   VAR
      sa_Parameter { ExternalAccessible := 'False'; ExternalVisible := 'False'; ExternalWritable := 'False'; S7_SetPoint := 'False'} : Array[1..16] of "UDT_VfdSinaParameterUser";   // Structure with parameters
      sa_ParameterEmpty { ExternalAccessible := 'False'; ExternalVisible := 'False'; ExternalWritable := 'False'; S7_SetPoint := 'False'} : Array[1..16] of "UDT_VfdSinaParameterUser";   // Empty structure
      sa_ParameterToCompare { ExternalAccessible := 'False'; ExternalVisible := 'False'; ExternalWritable := 'False'; S7_SetPoint := 'False'} : Array[1..16] of "UDT_VfdSinaParameterUser";   // Structure with parameters to compare
      sFB_SinaParaInstance {InstructionName := 'SinaPara'; LibVersion := '1.1'; ExternalAccessible := 'False'; ExternalVisible := 'False'; ExternalWritable := 'False'; S7_SetPoint := 'False'} : SinaPara;   // Write/read parameters to/from VFD
      sR_TRIG_StartJob {InstructionName := 'R_TRIG'; LibVersion := '1.0'; ExternalAccessible := 'False'; ExternalVisible := 'False'; ExternalWritable := 'False'; S7_SetPoint := 'False'} : R_TRIG;   // Bit for start trigger for rising edge
      sR_TRIG_Time {InstructionName := 'R_TRIG'; LibVersion := '1.0'; ExternalAccessible := 'False'; ExternalVisible := 'False'; ExternalWritable := 'False'; S7_SetPoint := 'False'} : R_TRIG;   // Bit for trigger for time couting
      sR_TRIG_DelayTime {InstructionName := 'R_TRIG'; LibVersion := '1.0'; ExternalAccessible := 'False'; ExternalVisible := 'False'; ExternalWritable := 'False'; S7_SetPoint := 'False'} : R_TRIG;   // Bit for trigger for time couting
      sF_TRIG_CancelJob {InstructionName := 'F_TRIG'; LibVersion := '1.0'; ExternalAccessible := 'False'; ExternalVisible := 'False'; ExternalWritable := 'False'; S7_SetPoint := 'False'} : F_TRIG;   // Bit for start trigger for falling edge
      sa_Status { ExternalAccessible := 'False'; ExternalVisible := 'False'; ExternalWritable := 'False'} : Struct   // Parametrization status
         StepNr { ExternalAccessible := 'False'; ExternalVisible := 'False'; ExternalWritable := 'False'} : Int;   // The number of the current step
         StepNrError { ExternalAccessible := 'False'; ExternalVisible := 'False'; ExternalWritable := 'False'} : Int;   // The number of the step in witch the error occurred
         ParameterNrError { ExternalAccessible := 'False'; ExternalVisible := 'False'; ExternalWritable := 'False'} : Int;   // The number of the parameter in witch the error occurred
         ResponseValueError { ExternalAccessible := 'False'; ExternalVisible := 'False'; ExternalWritable := 'False'} : Bool;   // Response value error
         WrongFormat { ExternalAccessible := 'False'; ExternalVisible := 'False'; ExternalWritable := 'False'} : Bool;   // Wrong parameter format
         TimeExceeded { ExternalAccessible := 'False'; ExternalVisible := 'False'; ExternalWritable := 'False'} : Bool;   // Time has been exceeded
         NeedAck { ExternalAccessible := 'False'; ExternalVisible := 'False'; ExternalWritable := 'False'} : Bool;   // Need acknowledge signal (to cintinue parametrization)
         StepDone { ExternalAccessible := 'False'; ExternalVisible := 'False'; ExternalWritable := 'False'} : Bool;   // Step done
         MemoryCardInserted { ExternalAccessible := 'False'; ExternalVisible := 'False'; ExternalWritable := 'False'} : Bool;   // The card is in the VFD, checked in step 51
      END_STRUCT;
      sa_SinaPara { ExternalAccessible := 'False'; ExternalVisible := 'False'; ExternalWritable := 'False'} : Struct   // Sina Para status
         DiagId { ExternalAccessible := 'False'; ExternalVisible := 'False'; ExternalWritable := 'False'} : Word;   // Expanded communication error
         ErrorId { ExternalAccessible := 'False'; ExternalVisible := 'False'; ExternalWritable := 'False'} : DWord;   // Error Id: 1st word (binary) coded as to which parameter access is faulted
         Error { ExternalAccessible := 'False'; ExternalVisible := 'False'; ExternalWritable := 'False'} : Bool;   // Main error signal from SINA_PARA instruction
      END_STRUCT;
      sa_Stepconfig { ExternalAccessible := 'False'; ExternalVisible := 'False'; ExternalWritable := 'False'} : Struct   // Structure with step configuration
         Read { ExternalAccessible := 'False'; ExternalVisible := 'False'; ExternalWritable := 'False'} : Bool;
         Write { ExternalAccessible := 'False'; ExternalVisible := 'False'; ExternalWritable := 'False'} : Bool;
         ParaNo { ExternalAccessible := 'False'; ExternalVisible := 'False'; ExternalWritable := 'False'} : Int;
         new_Step_config { ExternalAccessible := 'False'; ExternalVisible := 'False'; ExternalWritable := 'False'} : Struct
            Used { ExternalAccessible := 'False'; ExternalVisible := 'False'; ExternalWritable := 'False'} : Bool;
            Read { ExternalAccessible := 'False'; ExternalVisible := 'False'; ExternalWritable := 'False'} : Bool;
            Write { ExternalAccessible := 'False'; ExternalVisible := 'False'; ExternalWritable := 'False'} : Bool;
            ParaNo { ExternalAccessible := 'False'; ExternalVisible := 'False'; ExternalWritable := 'False'} : Int;
         END_STRUCT;
      END_STRUCT;
      sa_StepconfigEmpty { ExternalAccessible := 'False'; ExternalVisible := 'False'; ExternalWritable := 'False'} : Struct   // Empty structure
         Read { ExternalAccessible := 'False'; ExternalVisible := 'False'; ExternalWritable := 'False'} : Bool;
         Write { ExternalAccessible := 'False'; ExternalVisible := 'False'; ExternalWritable := 'False'} : Bool;
         ParaNo { ExternalAccessible := 'False'; ExternalVisible := 'False'; ExternalWritable := 'False'} : Int;
         new_Step_config { ExternalAccessible := 'False'; ExternalVisible := 'False'; ExternalWritable := 'False'} : Struct
            Used { ExternalAccessible := 'False'; ExternalVisible := 'False'; ExternalWritable := 'False'} : Bool;
            Read { ExternalAccessible := 'False'; ExternalVisible := 'False'; ExternalWritable := 'False'} : Bool;
            Write { ExternalAccessible := 'False'; ExternalVisible := 'False'; ExternalWritable := 'False'} : Bool;
            ParaNo { ExternalAccessible := 'False'; ExternalVisible := 'False'; ExternalWritable := 'False'} : Int;
         END_STRUCT;
      END_STRUCT;
      si_StepNr { ExternalAccessible := 'False'; ExternalVisible := 'False'; ExternalWritable := 'False'} : Int;   // Current step number
      si_StepNrOLD { ExternalAccessible := 'False'; ExternalVisible := 'False'; ExternalWritable := 'False'} : Int;   // Step number in previous PLC cycle
      si_StepTime { ExternalAccessible := 'False'; ExternalVisible := 'False'; ExternalWritable := 'False'} : Int;   // Step time
      si_DelayTime { ExternalAccessible := 'False'; ExternalVisible := 'False'; ExternalWritable := 'False'} : Int;   // The time after which is read the parameters
      si_StepNrError { ExternalAccessible := 'False'; ExternalVisible := 'False'; ExternalWritable := 'False'} : Int;   // The step number where the error is currently
      si_ParameterNrError { ExternalAccessible := 'False'; ExternalVisible := 'False'; ExternalWritable := 'False'} : Int;   // The parameter number where the error is currently
      si_SinaParaParaNo { ExternalAccessible := 'False'; ExternalVisible := 'False'; ExternalWritable := 'False'} : Int := 0;   // SinaPara- Number of parameter, 0 to 16
      si_Loop { ExternalAccessible := 'False'; ExternalVisible := 'False'; ExternalWritable := 'False'} : Int;   // Number of parameters used in loop
      sx_Only_motor_measuring { ExternalAccessible := 'False'; ExternalVisible := 'False'; ExternalWritable := 'False'} : Bool;   // [True] If the motor and VFD have been parameterized. Only measure the motor.
      sx_ActiveButtonGoToNextStep { ExternalAccessible := 'False'; ExternalVisible := 'False'; ExternalWritable := 'False'} : Bool;   // Button to go for the next step
      sx_Start { ExternalAccessible := 'False'; ExternalVisible := 'False'; ExternalWritable := 'False'} : Bool;   // Signal to start of parameterization function SinaPara
      sx_Busy { ExternalAccessible := 'False'; ExternalVisible := 'False'; ExternalWritable := 'False'} : Bool;   // Parametrization in progress (busy)
      sx_Done { ExternalAccessible := 'False'; ExternalVisible := 'False'; ExternalWritable := 'False'} : Bool;   // Parametrization done
      sx_Error { ExternalAccessible := 'False'; ExternalVisible := 'False'; ExternalWritable := 'False'} : Bool;   // Main error signal
      sx_OnlyRead { ExternalAccessible := 'False'; ExternalVisible := 'False'; ExternalWritable := 'False'} : Bool;   // Only read mode
      sx_OnlyWrite { ExternalAccessible := 'False'; ExternalVisible := 'False'; ExternalWritable := 'False'} : Bool;   // Only write mode
      sx_WriteRead { ExternalAccessible := 'False'; ExternalVisible := 'False'; ExternalWritable := 'False'} : Bool;   // Write and read mode
      sx_SinaParaStart { ExternalAccessible := 'False'; ExternalVisible := 'False'; ExternalWritable := 'False'} : Bool;   // SinaPara- Start of parameterization, 0= inactive function, 1= active function
      sx_SinaParaReadWrite { ExternalAccessible := 'False'; ExternalVisible := 'False'; ExternalWritable := 'False'} : Bool;   // SinaPara- Read/write parameters , 0=read parameter , 1=write parameter
      sx_SinaParaReady { ExternalAccessible := 'False'; ExternalVisible := 'False'; ExternalWritable := 'False'} : Bool;   // SinaPara- Ready to parameterization
      sx_SinaParaBusy { ExternalAccessible := 'False'; ExternalVisible := 'False'; ExternalWritable := 'False'} : Bool;   // SinaPara- Busy signal
      sx_SinaParaDone { ExternalAccessible := 'False'; ExternalVisible := 'False'; ExternalWritable := 'False'} : Bool;   // SinaPara- Parameterization done
      sx_ReadDone { ExternalAccessible := 'False'; ExternalVisible := 'False'; ExternalWritable := 'False'} : Bool;   // Read done
      sx_WriteDone { ExternalAccessible := 'False'; ExternalVisible := 'False'; ExternalWritable := 'False'} : Bool;   // Write done
      sx_PreparedData { ExternalAccessible := 'False'; ExternalVisible := 'False'; ExternalWritable := 'False'} : Bool;   // Step data prepared
      sx_TimeRTrig { ExternalAccessible := 'False'; ExternalVisible := 'False'; ExternalWritable := 'False'} : Bool;   // Trigger for time counting
      sx_ReadTime { ExternalAccessible := 'False'; ExternalVisible := 'False'; ExternalWritable := 'False'} : Bool;   // Read time, on this time the parameters are read in the loop
      sx_Freecycle { ExternalAccessible := 'False'; ExternalVisible := 'False'; ExternalWritable := 'False'} : Bool;   // "Empty" program cycle where the code is not executed, SinaPara need edge to start
      sx_StartMeasuring { ExternalAccessible := 'False'; ExternalVisible := 'False'; ExternalWritable := 'False'} : Bool;   // Start measuring
      sx_ComparisonParameters { ExternalAccessible := 'False'; ExternalVisible := 'False'; ExternalWritable := 'False'} : Bool;   // Comparison parameters ,1- Correct , 0- Bad
      sx_StartDelayTime { ExternalAccessible := 'False'; ExternalVisible := 'False'; ExternalWritable := 'False'} : Bool;   // Delay of reading parameters
      sx_ResponseValueError { ExternalAccessible := 'False'; ExternalVisible := 'False'; ExternalWritable := 'False'} : Bool;   // The parameter read out is not correct
      sx_WrongFormat { ExternalAccessible := 'False'; ExternalVisible := 'False'; ExternalWritable := 'False'} : Bool;   // The parameter has a wrong format
      sx_SelectedG120C { ExternalAccessible := 'False'; ExternalVisible := 'False'; ExternalWritable := 'False'} : Bool;   // Sequence from VFD G120C
      sx_SelectedG120D { ExternalAccessible := 'False'; ExternalVisible := 'False'; ExternalWritable := 'False'} : Bool;   // Sequence from VFD G120D
   END_VAR

   VAR CONSTANT
      cb_SinaParamAxisNo : Byte := 16#01;   // Axis number
      ci_StepTime : Int := 60;   // The time that the function has to read the correct parameters
   END_VAR


BEGIN
	(*
	----------------------------------------------------------------------------------------

	Version history:
	Date        | Version   | Author        | Remark
	----------------------------------------------------------------------------------------
	24/06/2019  | 1.0       | S. Nikodem    | first release MHS TIA 15.1
	12/11/2019  | 3.0       | P. Majka      | 3.0 MHS library release TIA 15.1
	12/10/2021  | 3.2       | S. Nikodem    | new release MHS TIA 15.1
	03/11/2021  | 3.3       | M. Piela      | Add comments
	21/02/2023  | 4.0       | F.Baten       | 4.0 Release TIA 17.5
	*)

	REGION 1 - Start Job

	    // Monitor rising trigger if is input enable signal
	    #sR_TRIG_StartJob(CLK := #ix_Enable);

	    // If start trigger  occurs for a rising edge then variables to start conditions are prepared
	    IF (#sR_TRIG_StartJob.Q)
	    THEN

	        #sx_Start := TRUE;
	        #sx_Busy := TRUE;
	        #sx_Done := FALSE;
	        #sx_Error := FALSE;
	        #sx_Freecycle := FALSE;
	        #sx_ReadDone := FALSE;
	        #sx_WriteDone := FALSE;
	        #sx_PreparedData := FALSE;
	        #si_StepTime := 0;
	        #sx_ResponseValueError := FALSE;
	        #sx_WrongFormat := FALSE;
	        #si_StepNrError := 0;
	        #si_ParameterNrError := 0;
	        #sx_StartDelayTime := FALSE;
	        #sa_Status.MemoryCardInserted := FALSE;

	        #sa_Status.StepDone := FALSE;
	        #sa_Status.NeedAck := FALSE;
	        #sa_Status.ResponseValueError := FALSE;
	        #sa_Status.StepNrError := 0;
	        #sa_Status.ParameterNrError := 0;
	        #sa_Status.TimeExceeded := FALSE;

	        #si_StepNr := 1;

	        //After activation bit “sx_Only_motor_measuring” sequence jump to step 44 and only the motor measurement
	        //and all steps after it will be performed. But before that VFD, Safety must be configured and switched on 400 V.
	        IF #sx_Only_motor_measuring THEN

	            #si_StepNr := 44;

	        END_IF;

	    END_IF;

	END_REGION

	REGION 2 - Cancel Job

	    // Monitor falling trigger if is input enable signal
	    #sF_TRIG_CancelJob(CLK := #ix_Enable);

	    // If occurs start trigger for falling edge
	    IF (#sF_TRIG_CancelJob.Q)
	    THEN

	        #sx_Start := FALSE;
	        #sx_Busy := FALSE;
	        #sx_StartMeasuring := FALSE;

	        // If parametrization is not done
	        IF (NOT #sx_Done)
	        THEN

	            #sx_Error := TRUE;

	        END_IF;

	    END_IF;

	END_REGION

	REGION 3 - Clean structure

	    //When a step in the sequence changes, the structure must be cleared
	    IF (#si_StepNrOLD <> #si_StepNr) OR #sR_TRIG_StartJob.Q THEN

	        #sa_Parameter := #sa_ParameterEmpty;
	        #sa_Stepconfig := #sa_StepconfigEmpty;

	    END_IF;

	    //Copy step number
	    #si_StepNrOLD := #si_StepNr;

	END_REGION

	REGION 4 - Sequence steps

	    //The VFD type is selected based on the variable "# i_UDT_MotorConfig.VFDType"
	    #sx_SelectedG120D := #iUDT_MotorConfig.VFDType = 5302 OR
	    #iUDT_MotorConfig.VFDType = 5304 OR
	    #iUDT_MotorConfig.VFDType = 5306 OR
	    #iUDT_MotorConfig.VFDType = 5307 OR
	    #iUDT_MotorConfig.VFDType = 5308 OR
	    #iUDT_MotorConfig.VFDType = 5309;

	    #sx_SelectedG120C := #iUDT_MotorConfig.VFDType = 1;

	    REGION Step 1

	        IF #si_StepNr = 1 THEN

	            //Step configuration
	            #sa_Stepconfig.Read := TRUE;           //Paramerters are readed
	            #sa_Stepconfig.Write := TRUE;          //Paramerters are write
	            #sa_Stepconfig.ParaNo := 1;            //Defined how many parameters are used

	            //Used parameters in this step
	            //1 - Drive commissioning mode, 30: Parameter reset
	            #sa_Parameter[1].siParaNo := 10;        //Parameter number
	            #sa_Parameter[1].srValue := 30.0;       //Parameter value
	            #sa_Parameter[1].syFormat := 3;         //Parameter format

	        END_IF;

	    END_REGION

	    REGION Step 2

	        IF #si_StepNr = 2 THEN

	            //Step configuration
	            #sa_Stepconfig.Write := TRUE;
	            #sa_Stepconfig.ParaNo := 1;

	            //Used parameters in this step
	            //1 - Reset drive parameters, 1: Start a parameter reset
	            #sa_Parameter[1].siParaNo := 970;
	            #sa_Parameter[1].srValue := 1.0;
	            #sa_Parameter[1].syFormat := 16#0006;

	        END_IF;

	    END_REGION

	    REGION Step 3

	        IF #si_StepNr = 3 THEN

	            //Step configuration
	            #sa_Stepconfig.Read := TRUE;
	            #sa_Stepconfig.ParaNo := 3;

	            //Used parameters in this step
	            //1 - Drive commissioning mode, 1: Quick commissioning
	            #sa_Parameter[1].siParaNo := 10;
	            #sa_Parameter[1].srValue := 1.0;
	            #sa_Parameter[1].syFormat := 16#0003;
	            //2 - Reset drive parameters
	            #sa_Parameter[2].siParaNo := 970;
	            #sa_Parameter[2].syFormat := 16#0006;
	            //3 - Parameter write inhibit status
	            #sa_Parameter[3].siParaNo := 3996;
	            #sa_Parameter[3].syFormat := 0;

	        END_IF;

	    END_REGION

	    REGION Step 4

	        IF #si_StepNr = 4 THEN

	            //Step configuration
	            #sa_Stepconfig.Read := TRUE;
	            #sa_Stepconfig.Write := TRUE;
	            #sa_Stepconfig.ParaNo := 1;

	            //Used parameters in this step
	            //1 - Drive commissioning mode, 30: Parameter reset
	            #sa_Parameter[1].siParaNo := 10;
	            #sa_Parameter[1].srValue := 30.0;
	            #sa_Parameter[1].syFormat := 3;

	        END_IF;

	    END_REGION

	    REGION Step 5

	        IF #si_StepNr = 5 THEN

	            //Step configuration
	            #sa_Stepconfig.Write := TRUE;
	            #sa_Stepconfig.ParaNo := 2;

	            //Used parameters in this step
	            //1 - SI password input, 0 = default value
	            #sa_Parameter[1].siParaNo := 9761;
	            #sa_Parameter[1].syFormat := 7;
	            //2 - Drive commissioning mode, 30: Parameter reset
	            #sa_Parameter[2].siParaNo := 10;
	            #sa_Parameter[2].srValue := 30.0;
	            #sa_Parameter[2].syFormat := 3;

	        END_IF;

	    END_REGION

	    REGION Step 6

	        IF #si_StepNr = 6 THEN

	            //Step configuration
	            #sa_Stepconfig.Read := TRUE;
	            #sa_Stepconfig.Write := TRUE;
	            #sa_Stepconfig.ParaNo := 1;

	            //Used parameters in this step
	            //1 - Reset drive parameters, 5: Starts a safety parameter reset
	            #sa_Parameter[1].siParaNo := 970;
	            #sa_Parameter[1].srValue := 5.0;
	            #sa_Parameter[1].syFormat := 3;

	        END_IF;

	    END_REGION

	    REGION Step 7

	        IF #si_StepNr = 7 THEN

	            //Step configuration
	            #sa_Stepconfig.Read := TRUE;
	            #sa_Stepconfig.ParaNo := 3;

	            //Used parameters in this step
	            //1 - Drive commissioning mode, 1: Quick commissioning
	            #sa_Parameter[1].siParaNo := 10;
	            #sa_Parameter[1].srValue := 1.0;
	            #sa_Parameter[1].syFormat := 3;
	            //2 - Reset drive parameters
	            #sa_Parameter[2].siParaNo := 970;
	            #sa_Parameter[2].syFormat := BYTE#16#03;
	            //3 - Parameter write inhibit status
	            #sa_Parameter[3].siParaNo := 3996;
	            #sa_Parameter[3].syFormat := BYTE#16#05;

	        END_IF;

	    END_REGION

	    REGION Step 8

	        IF #si_StepNr = 8 THEN

	            //Step configuration
	            #sa_Stepconfig.Write := TRUE;
	            #sa_Stepconfig.ParaNo := 1;

	            //Used parameters in this step
	            //1 - Save parameters, 1: Save drive object
	            #sa_Parameter[1].siParaNo := 971;
	            #sa_Parameter[1].srValue := 1.0;
	            #sa_Parameter[1].syFormat := 6;

	        END_IF;

	    END_REGION

	    REGION Step 9

	        IF #si_StepNr = 9 THEN

	            //Step configuration
	            #sa_Stepconfig.Read := TRUE;
	            #sa_Stepconfig.ParaNo := 1;

	            //Used parameters in this step
	            //1 - Save parameters
	            #sa_Parameter[1].siParaNo := 971;
	            #sa_Parameter[1].syFormat := 6;

	        END_IF;

	    END_REGION

	    REGION Step 10

	        IF #si_StepNr = 10 THEN

	            //Step configuration
	            #sa_Stepconfig.Read := TRUE;
	            #sa_Stepconfig.Write := TRUE;
	            #sa_Stepconfig.ParaNo := 1;

	            //Used parameters in this step
	            //1 - Drive commissioning mode, 1: Quick commissioning
	            #sa_Parameter[1].siParaNo := 10;
	            #sa_Parameter[1].srValue := 1.0;
	            #sa_Parameter[1].syFormat := 3;

	        END_IF;

	    END_REGION

	    REGION Step 11

	        IF #si_StepNr = 11 AND #sx_SelectedG120D THEN

	            //Step configuration
	            #sa_Stepconfig.Read := TRUE;
	            #sa_Stepconfig.Write := TRUE;
	            #sa_Stepconfig.ParaNo := 8;

	            //Used parameters in this step
	            //1 - Macro drive unit
	            #sa_Parameter[1].siParaNo := 15;
	            #sa_Parameter[1].sdValue := 27;
	            #sa_Parameter[1].syFormat := BYTE#16#07;
	            //2 - Power unit application
	            #sa_Parameter[2].siParaNo := 205;
	            #sa_Parameter[2].syFormat := BYTE#16#03;
	            //3 - Automatic calculation motor/control parameters
	            #sa_Parameter[3].siParaNo := 340;
	            #sa_Parameter[3].syFormat := BYTE#16#03;
	            //4 - Technology application
	            #sa_Parameter[4].siParaNo := 500;
	            #sa_Parameter[4].syFormat := BYTE#16#03;
	            //5 - Field bus interface protocol selection
	            #sa_Parameter[5].siParaNo := 2030;
	            #sa_Parameter[5].srValue := 7.0;
	            #sa_Parameter[5].syFormat := BYTE#16#03;
	            //6 - IEC/NEMA mot stds
	            #sa_Parameter[6].siParaNo := 100;
	            #sa_Parameter[6].syFormat := BYTE#16#03;
	            //7 - Drive filter type motor side
	            #sa_Parameter[7].siParaNo := 230;
	            #sa_Parameter[7].syFormat := BYTE#16#03;
	            //8 - Motor cooling type
	            #sa_Parameter[8].siParaNo := 335;
	            #sa_Parameter[8].syFormat := BYTE#16#03;

	        END_IF;

	        IF #si_StepNr = 11 AND #sx_SelectedG120C THEN

	            //Step configuration
	            #sa_Stepconfig.Read := TRUE;
	            #sa_Stepconfig.Write := TRUE;
	            #sa_Stepconfig.ParaNo := 6;

	            //Used parameters in this step
	            //1 - Macro drive unit
	            #sa_Parameter[1].siParaNo := 15;
	            #sa_Parameter[1].sdValue := 7;
	            #sa_Parameter[1].syFormat := BYTE#16#07;
	            //2 - Automatic calculation motor/control parameters
	            #sa_Parameter[2].siParaNo := 340;
	            #sa_Parameter[2].syFormat := BYTE#16#03;
	            //3 - Field bus interface protocol selection
	            #sa_Parameter[3].siParaNo := 2030;
	            #sa_Parameter[3].srValue := 7.0;
	            #sa_Parameter[3].syFormat := BYTE#16#03;
	            //4 - IEC/NEMA mot stds
	            #sa_Parameter[4].siParaNo := 100;
	            #sa_Parameter[4].syFormat := BYTE#16#03;
	            //5 - Drive filter type motor side
	            #sa_Parameter[5].siParaNo := 230;
	            #sa_Parameter[5].syFormat := BYTE#16#03;
	            //6 - Motor cooling type
	            #sa_Parameter[6].siParaNo := 335;
	            #sa_Parameter[6].syFormat := BYTE#16#03;

	        END_IF;

	    END_REGION

	    REGION Step 12

	        IF #si_StepNr = 12 AND #sx_SelectedG120D THEN

	            //Step configuration
	            #sa_Stepconfig.Read := TRUE;
	            #sa_Stepconfig.Write := TRUE;
	            #sa_Stepconfig.ParaNo := 1;

	            //Used parameters in this step
	            //1 - Open-loop/closed-loop control operating mode
	            IF #iUDT_MotorConfig.EncoderConfig THEN

	                #sa_Parameter[1].siParaNo := 1300;
	                #sa_Parameter[1].srValue := 21.0;           //21: Speed control (with encoder)
	                #sa_Parameter[1].syFormat := BYTE#16#03;

	            ELSE

	                #sa_Parameter[1].siParaNo := 1300;
	                #sa_Parameter[1].srValue := 20.0;           //20: Speed control (encoderless)
	                #sa_Parameter[1].syFormat := BYTE#16#03;

	            END_IF;

	        END_IF;

	        IF #si_StepNr = 12 AND #sx_SelectedG120C THEN

	            //Step configuration
	            #sa_Stepconfig.Read := TRUE;
	            #sa_Stepconfig.Write := TRUE;
	            #sa_Stepconfig.ParaNo := 1;

	            //Used parameters in this step
	            //1 - PROFIdrive PZD telegram selection, 999: Free telegram configuration with BICO
	            #sa_Parameter[1].siParaNo := 922;
	            #sa_Parameter[1].srValue := 999.0;
	            #sa_Parameter[1].syFormat := BYTE#16#06;

	        END_IF;

	    END_REGION

	    REGION Step 13

	        IF #si_StepNr = 13 THEN

	            //Step configuration
	            #sa_Stepconfig.Read := TRUE;
	            #sa_Stepconfig.Write := TRUE;
	            #sa_Stepconfig.ParaNo := 3;

	            //Used parameters in this step
	            //1 - PROFIdrive PZD telegram selection, 999: Free telegram configuration with BICO
	            #sa_Parameter[1].siParaNo := 922;
	            #sa_Parameter[1].srValue := 999.0;
	            #sa_Parameter[1].syFormat := BYTE#16#06;
	            //2 - Speed setpoint selection, 6: No supplementary setpoint + Fieldbus
	            #sa_Parameter[2].siParaNo := 1000;
	            #sa_Parameter[2].srValue := 6.0;
	            #sa_Parameter[2].syFormat := BYTE#16#03;
	            //3 - Motor data identification and rotating measurement
	            #sa_Parameter[3].siParaNo := 1900;
	            #sa_Parameter[3].syFormat := 16#0003;
	            #sa_Parameter[3].swErrorNo := 16#0000;

	        END_IF;

	    END_REGION

	    REGION Step 14

	        IF #si_StepNr = 14 THEN

	            //Step configuration
	            #sa_Stepconfig.Read := TRUE;
	            #sa_Stepconfig.Write := TRUE;
	            #sa_Stepconfig.ParaNo := 16;

	            //Used parameters in this step
	            //1 - Telegram word 1 bit 0
	            #sa_Parameter[1].siParaNo := 2080;
	            #sa_Parameter[1].sdValue := 58981376;       //r899.0
	            #sa_Parameter[1].syFormat := BYTE#16#07;
	            //2 - Telegram word 1 bit 1
	            #sa_Parameter[2].siParaNo := 2080;
	            #sa_Parameter[2].siIndex := 1;
	            #sa_Parameter[2].sdValue := 58981377;       //r899.1
	            #sa_Parameter[2].syFormat := BYTE#16#07;
	            //3 - Telegram word 1 bit 2
	            #sa_Parameter[3].siParaNo := 2080;
	            #sa_Parameter[3].siIndex := 2;
	            #sa_Parameter[3].sdValue := 58981378;       //r899.2
	            #sa_Parameter[3].syFormat := BYTE#16#07;
	            //4 - Telegram word 1 bit 3
	            #sa_Parameter[4].siParaNo := 2080;
	            #sa_Parameter[4].siIndex := 3;
	            #sa_Parameter[4].sdValue := 140_246_019;    //r2139.3
	            #sa_Parameter[4].syFormat := BYTE#16#07;
	            //5 - Telegram word 1 bit 4
	            #sa_Parameter[5].siParaNo := 2080;
	            #sa_Parameter[5].siIndex := 4;
	            #sa_Parameter[5].sdValue := 58981380;       //r899.4
	            #sa_Parameter[5].syFormat := BYTE#16#07;
	            //6 - Telegram word 1 bit 5
	            #sa_Parameter[6].siParaNo := 2080;
	            #sa_Parameter[6].siIndex := 5;
	            #sa_Parameter[6].sdValue := 58981381;       //r889.5
	            #sa_Parameter[6].syFormat := BYTE#16#07;
	            //7 - Telegram word 1 bit 6
	            #sa_Parameter[7].siParaNo := 2080;
	            #sa_Parameter[7].siIndex := 6;
	            #sa_Parameter[7].syFormat := BYTE#16#07;
	            //8 - Telegram word 1 bit 7
	            #sa_Parameter[8].siParaNo := 2080;
	            #sa_Parameter[8].siIndex := 7;
	            #sa_Parameter[8].sdValue := 140_246_023;        //r2139.7
	            #sa_Parameter[8].syFormat := BYTE#16#07;
	            //9 - Telegram word 1 bit 8
	            #sa_Parameter[9].siParaNo := 2080;
	            #sa_Parameter[9].siIndex := 8;
	            #sa_Parameter[9].syFormat := BYTE#16#07;
	            //10 - Telegram word 1 bit 9
	            #sa_Parameter[10].siParaNo := 2080;
	            #sa_Parameter[10].siIndex := 9;
	            #sa_Parameter[10].sdValue := 58981385;          //r899.9
	            #sa_Parameter[10].syFormat := BYTE#16#07;
	            //11 - Telegram word 1 bit 10
	            #sa_Parameter[11].siParaNo := 2080;
	            #sa_Parameter[11].siIndex := 10;
	            #sa_Parameter[11].syFormat := BYTE#16#07;
	            //12 - Telegram word 1 bit 11
	            #sa_Parameter[12].siParaNo := 2080;
	            #sa_Parameter[12].siIndex := 11;
	            #sa_Parameter[12].syFormat := BYTE#16#07;
	            //13 - Telegram word 1 bit 12
	            #sa_Parameter[13].siParaNo := 2080;
	            #sa_Parameter[13].siIndex := 12;
	            #sa_Parameter[13].sdValue := 58981388;          //r899.12
	            #sa_Parameter[13].syFormat := BYTE#16#07;
	            //14 - Telegram word 1 bit 13
	            #sa_Parameter[14].siParaNo := 2080;
	            #sa_Parameter[14].siIndex := 13;
	            #sa_Parameter[14].sdValue := 139_983_886;       //r2135.14
	            #sa_Parameter[14].syFormat := BYTE#16#07;
	            //15 - Telegram word 1 bit 14
	            #sa_Parameter[15].siParaNo := 2080;
	            #sa_Parameter[15].siIndex := 14;
	            #sa_Parameter[15].sdValue := 144_047_107;       //r2197.3
	            #sa_Parameter[15].syFormat := BYTE#16#07;
	            //16 - Telegram word 1 bit 15
	            #sa_Parameter[16].siParaNo := 2080;
	            #sa_Parameter[16].siIndex := 15;
	            #sa_Parameter[16].sdValue := 139_983_887;       //r2135.15
	            #sa_Parameter[16].syFormat := BYTE#16#07;

	        END_IF;

	    END_REGION

	    REGION Step 15

	        IF #si_StepNr = 15 AND #sx_SelectedG120D THEN

	            //Step configuration
	            #sa_Stepconfig.Read := TRUE;
	            #sa_Stepconfig.Write := TRUE;
	            #sa_Stepconfig.ParaNo := 15;

	            //Used parameters in this step
	            //1 - Invert binector-connector converter status word
	            #sa_Parameter[1].siParaNo := 2088;
	            #sa_Parameter[1].srValue := 43008.0;
	            #sa_Parameter[1].syFormat := BYTE#16#06;

	            //CI: PROFIdrive PZD send word
	            //2 - Telegram word 0
	            #sa_Parameter[2].siParaNo := 2051;
	            #sa_Parameter[2].sdValue := 136_969_216;
	            #sa_Parameter[2].syFormat := BYTE#16#07;
	            //3 - Telegram word 1
	            #sa_Parameter[3].siParaNo := 2051;
	            #sa_Parameter[3].siIndex := 1;
	            #sa_Parameter[3].sdValue := 4193280;
	            #sa_Parameter[3].syFormat := BYTE#16#07;
	            //4 - Telegram word 2
	            #sa_Parameter[4].siParaNo := 2051;
	            #sa_Parameter[4].siIndex := 2;
	            #sa_Parameter[4].sdValue := 4520961;
	            #sa_Parameter[4].syFormat := BYTE#16#07;
	            //5 - Telegram word 3
	            #sa_Parameter[5].siParaNo := 2051;
	            #sa_Parameter[5].siIndex := 3;
	            #sa_Parameter[5].sdValue := 5307393;
	            #sa_Parameter[5].syFormat := BYTE#16#07;
	            //6 - Telegram word 4
	            #sa_Parameter[6].siParaNo := 2051;
	            #sa_Parameter[6].siIndex := 4;
	            #sa_Parameter[6].sdValue := 139_787_264;
	            #sa_Parameter[6].syFormat := BYTE#16#07;
	            //7 - Telegram word 5
	            #sa_Parameter[7].siParaNo := 2051;
	            #sa_Parameter[7].siIndex := 5;
	            #sa_Parameter[7].sdValue := 139_721_728;
	            #sa_Parameter[7].syFormat := BYTE#16#07;
	            //8 - Telegram word 9
	            #sa_Parameter[8].siParaNo := 2051;
	            #sa_Parameter[8].siIndex := 9;
	            #sa_Parameter[8].syFormat := BYTE#16#07;
	            //9 - Telegram word 10
	            #sa_Parameter[9].siParaNo := 2051;
	            #sa_Parameter[9].siIndex := 10;
	            #sa_Parameter[9].syFormat := BYTE#16#07;
	            //10 - Telegram word 11
	            #sa_Parameter[10].siParaNo := 2051;
	            #sa_Parameter[10].siIndex := 11;
	            #sa_Parameter[10].sdValue := 47381504;
	            #sa_Parameter[10].syFormat := BYTE#16#07;

	            //CI: PROFIdrive PZD send double word
	            //11 - Telegrm double word 5
	            #sa_Parameter[11].siParaNo := 2061;
	            #sa_Parameter[11].siIndex := 5;
	            #sa_Parameter[11].syFormat := BYTE#16#07;
	            //12 - Telegrm double word 6
	            #sa_Parameter[12].siParaNo := 2061;
	            #sa_Parameter[12].siIndex := 6;
	            #sa_Parameter[12].syFormat := BYTE#16#07;
	            //13 - Telegrm double word 7
	            #sa_Parameter[13].siParaNo := 2061;
	            #sa_Parameter[13].siIndex := 7;
	            #sa_Parameter[13].syFormat := BYTE#16#07;

	            //14 - CI: Ramp-function generator ramp-up time scaling
	            #sa_Parameter[14].siParaNo := 1138;
	            #sa_Parameter[14].sdValue := 134_413_314;
	            #sa_Parameter[14].syFormat := BYTE#16#07;
	            //15 - CI: Ramp-function generator ramp-down time scaling
	            #sa_Parameter[15].siParaNo := 1139;
	            #sa_Parameter[15].sdValue := 134_413_315;
	            #sa_Parameter[15].syFormat := BYTE#16#07;

	        END_IF;

	        IF #si_StepNr = 15 AND #sx_SelectedG120C THEN

	            //Step configuration
	            #sa_Stepconfig.Read := TRUE;
	            #sa_Stepconfig.Write := TRUE;
	            #sa_Stepconfig.ParaNo := 14;

	            //Used parameters in this step
	            //1 - Invert binector-connector converter status word
	            #sa_Parameter[1].siParaNo := 2088;
	            #sa_Parameter[1].srValue := 43008.0;
	            #sa_Parameter[1].syFormat := BYTE#16#06;
	            //2 - CI: PROFIdrive PZD send word
	            #sa_Parameter[2].siParaNo := 2051;
	            #sa_Parameter[2].sdValue := 136_969_216;
	            #sa_Parameter[2].syFormat := BYTE#16#07;
	            //3 - Telegram word 1
	            #sa_Parameter[3].siParaNo := 2051;
	            #sa_Parameter[3].siIndex := 1;
	            #sa_Parameter[3].sdValue := 4193280;
	            #sa_Parameter[3].syFormat := BYTE#16#07;
	            //4 - Telegram word 2
	            #sa_Parameter[4].siParaNo := 2051;
	            #sa_Parameter[4].siIndex := 2;
	            #sa_Parameter[4].sdValue := 4520961;
	            #sa_Parameter[4].syFormat := BYTE#16#07;
	            //5 - Telegram word 3
	            #sa_Parameter[5].siParaNo := 2051;
	            #sa_Parameter[5].siIndex := 3;
	            #sa_Parameter[5].sdValue := 5307393;
	            #sa_Parameter[5].syFormat := BYTE#16#07;
	            //6 - Telegram word 4
	            #sa_Parameter[6].siParaNo := 2051;
	            #sa_Parameter[6].siIndex := 4;
	            #sa_Parameter[6].sdValue := 139_787_264;
	            #sa_Parameter[6].syFormat := BYTE#16#07;
	            //7 - Telegram word 11
	            #sa_Parameter[7].siParaNo := 2051;
	            #sa_Parameter[7].siIndex := 11;
	            #sa_Parameter[7].sdValue := 47381504;
	            #sa_Parameter[7].syFormat := BYTE#16#07;
	            //8 - Telegram word 9
	            #sa_Parameter[8].siParaNo := 2051;
	            #sa_Parameter[8].siIndex := 9;
	            #sa_Parameter[8].syFormat := BYTE#16#07;
	            //9 - Telegram word 10
	            #sa_Parameter[9].siParaNo := 2051;
	            #sa_Parameter[9].siIndex := 10;
	            #sa_Parameter[9].syFormat := BYTE#16#07;
	            //CI: PROFIdrive PZD send double word
	            //10 - Telegrm double word 5
	            #sa_Parameter[10].siParaNo := 2061;
	            #sa_Parameter[10].siIndex := 5;
	            #sa_Parameter[10].syFormat := BYTE#16#07;
	            //11 - Telegrm double word 6
	            #sa_Parameter[11].siParaNo := 2061;
	            #sa_Parameter[11].siIndex := 6;
	            #sa_Parameter[11].syFormat := BYTE#16#07;
	            //12 - Telegrm double word 5
	            #sa_Parameter[12].siParaNo := 2061;
	            #sa_Parameter[12].siIndex := 5;
	            #sa_Parameter[12].syFormat := BYTE#16#08;
	            //13 - CI: Ramp-function generator ramp-up time scaling
	            #sa_Parameter[13].siParaNo := 1138;
	            #sa_Parameter[13].sdValue := 134_413_314;
	            #sa_Parameter[13].syFormat := BYTE#16#07;
	            //14 - CI: Ramp-function generator ramp-down time scaling
	            #sa_Parameter[14].siParaNo := 1139;
	            #sa_Parameter[14].sdValue := 134_413_315;
	            #sa_Parameter[14].syFormat := BYTE#16#07;


	        END_IF;

	    END_REGION

	    REGION Step 16

	        IF #si_StepNr = 16 AND #sx_SelectedG120D THEN

	            //Step configuration
	            #sa_Stepconfig.Read := TRUE;
	            #sa_Stepconfig.Write := TRUE;
	            #sa_Stepconfig.ParaNo := 14;

	            //Used parameters in this step
	            //1 - BI: ON/OFF (OFF1)
	            #sa_Parameter[1].siParaNo := 840;
	            #sa_Parameter[1].sdValue := 137_034_752;
	            #sa_Parameter[1].syFormat := BYTE#16#07;
	            //2 - BI: No coast-down / coast-down (OFF2) signal source 1
	            #sa_Parameter[2].siParaNo := 844;
	            #sa_Parameter[2].sdValue := 137_034_753;
	            #sa_Parameter[2].syFormat := BYTE#16#07;
	            //3 - BI: No Quick Stop / Quick Stop (OFF3) signal source 1
	            #sa_Parameter[3].siParaNo := 848;
	            #sa_Parameter[3].sdValue := 137_034_754;
	            #sa_Parameter[3].syFormat := BYTE#16#07;
	            //4 - BI: Enable operation/inhibit operation
	            #sa_Parameter[4].siParaNo := 852;
	            #sa_Parameter[4].sdValue := 137_034_755;
	            #sa_Parameter[4].syFormat := BYTE#16#07;
	            //5 - BI: Enable ramp-function generator/inhibit ramp-function generator
	            #sa_Parameter[5].siParaNo := 1140;
	            #sa_Parameter[5].sdValue := 137_034_756;
	            #sa_Parameter[5].syFormat := BYTE#16#07;
	            //6 - BI: Continue ramp-function generator/freeze ramp-function generator
	            #sa_Parameter[6].siParaNo := 1141;
	            #sa_Parameter[6].sdValue := 137_034_757;
	            #sa_Parameter[6].syFormat := BYTE#16#07;
	            //7 - BI: Enable setpoint/inhibit setpoint
	            #sa_Parameter[7].siParaNo := 1142;
	            #sa_Parameter[7].sdValue := 137_034_758;
	            #sa_Parameter[7].syFormat := BYTE#16#07;
	            //8 - BI: 1st acknowledge faults
	            #sa_Parameter[8].siParaNo := 2103;
	            #sa_Parameter[8].sdValue := 137_034_759;
	            #sa_Parameter[8].syFormat := BYTE#16#07;
	            //9 - BI: Control by PLC/no control by PLC
	            #sa_Parameter[9].siParaNo := 854;
	            #sa_Parameter[9].sdValue := 137_034_762;
	            #sa_Parameter[9].syFormat := BYTE#16#07;
	            //10 - BI: Setpoint inversion
	            #sa_Parameter[10].siParaNo := 1113;
	            #sa_Parameter[10].sdValue := 137_034_763;
	            #sa_Parameter[10].syFormat := BYTE#16#07;
	            //11 - CI: Main setpoint
	            #sa_Parameter[11].siParaNo := 1070;
	            #sa_Parameter[11].sdValue := 134_413_313;
	            #sa_Parameter[11].syFormat := BYTE#16#07;
	            //12 - CI: Connector-binector converter signal source
	            #sa_Parameter[12].siParaNo := 2099;
	            #sa_Parameter[12].sdValue := 134_413_323;
	            #sa_Parameter[12].syFormat := BYTE#16#07;
	            //13 - BI: CU signal source for terminal DO 0
	            #sa_Parameter[13].siParaNo := 730;
	            #sa_Parameter[13].sdValue := 137_296_896;
	            #sa_Parameter[13].syFormat := BYTE#16#07;
	            //14 - BI: CU signal source for terminal DO 1
	            #sa_Parameter[14].siParaNo := 731;
	            #sa_Parameter[14].sdValue := 137_296_897;
	            #sa_Parameter[14].syFormat := BYTE#16#07;

	        END_IF;

	        IF #si_StepNr = 16 AND #sx_SelectedG120C THEN

	            //Step configuration
	            #sa_Stepconfig.Read := TRUE;
	            #sa_Stepconfig.Write := TRUE;
	            #sa_Stepconfig.ParaNo := 15;

	            //Used parameters in this step
	            //1 - BI: ON/OFF (OFF1)
	            #sa_Parameter[1].siParaNo := 840;
	            #sa_Parameter[1].sdValue := 137_034_752;
	            #sa_Parameter[1].syFormat := BYTE#16#07;
	            //2 - BI: No coast-down / coast-down (OFF2) signal source 1
	            #sa_Parameter[2].siParaNo := 844;
	            #sa_Parameter[2].sdValue := 137_034_753;
	            #sa_Parameter[2].syFormat := BYTE#16#07;
	            //3 - BI: No Quick Stop / Quick Stop (OFF3) signal source 1
	            #sa_Parameter[3].siParaNo := 848;
	            #sa_Parameter[3].sdValue := 137_034_754;
	            #sa_Parameter[3].syFormat := BYTE#16#07;
	            //4 - BI: Enable operation/inhibit operation
	            #sa_Parameter[4].siParaNo := 852;
	            #sa_Parameter[4].sdValue := 137_034_755;
	            #sa_Parameter[4].syFormat := BYTE#16#07;
	            //5 - BI: Enable ramp-function generator/inhibit ramp-function generator
	            #sa_Parameter[5].siParaNo := 1140;
	            #sa_Parameter[5].sdValue := 137_034_756;
	            #sa_Parameter[5].syFormat := BYTE#16#07;
	            //6 - BI: Continue ramp-function generator/freeze ramp-function generator
	            #sa_Parameter[6].siParaNo := 1141;
	            #sa_Parameter[6].sdValue := 137_034_757;
	            #sa_Parameter[6].syFormat := BYTE#16#07;
	            //7 - BI: Enable setpoint/inhibit setpoint
	            #sa_Parameter[7].siParaNo := 1142;
	            #sa_Parameter[7].sdValue := 137_034_758;
	            #sa_Parameter[7].syFormat := BYTE#16#07;
	            //8 - BI: 1st acknowledge faults
	            #sa_Parameter[8].siParaNo := 2103;
	            #sa_Parameter[8].sdValue := 137_034_759;
	            #sa_Parameter[8].syFormat := BYTE#16#07;
	            //9 - BI: Control by PLC/no control by PLC
	            #sa_Parameter[9].siParaNo := 854;
	            #sa_Parameter[9].sdValue := 137_034_762;
	            #sa_Parameter[9].syFormat := BYTE#16#07;
	            //10 - BI: Setpoint inversion
	            #sa_Parameter[10].siParaNo := 1113;
	            #sa_Parameter[10].sdValue := 137_034_763;
	            #sa_Parameter[10].syFormat := BYTE#16#07;
	            //11 - CI: Main setpoint
	            #sa_Parameter[11].siParaNo := 1070;
	            #sa_Parameter[11].sdValue := 134_413_313;
	            #sa_Parameter[11].syFormat := BYTE#16#07;
	            //12 - CI: Connector-binector converter signal source
	            #sa_Parameter[12].siParaNo := 2099;
	            #sa_Parameter[12].sdValue := 134_413_323;
	            #sa_Parameter[12].syFormat := BYTE#16#07;
	            //13 - BI: CU signal source for terminal DO 0
	            #sa_Parameter[13].siParaNo := 730;
	            #sa_Parameter[13].sdValue := 3472387;
	            #sa_Parameter[13].syFormat := BYTE#16#07;

	            IF #iUDT_MotorConfig.BrakeConfig THEN

	                //14 - BI: CU signal source for terminal DO 1
	                #sa_Parameter[14].siParaNo := 731;
	                #sa_Parameter[14].sdValue := 58981388;
	                #sa_Parameter[14].syFormat := BYTE#16#07;

	            ELSE

	                //14 - BI: CU signal source for terminal DO 1
	                #sa_Parameter[14].siParaNo := 731;
	                #sa_Parameter[14].sdValue := 3537922;
	                #sa_Parameter[14].syFormat := BYTE#16#07;

	            END_IF;

	            //CI: PROFIdrive PZD send word
	            //15 - Telegram word 5
	            #sa_Parameter[15].siParaNo := 2051;
	            #sa_Parameter[15].siIndex := 5;
	            #sa_Parameter[15].sdValue := 139_721_728;
	            #sa_Parameter[15].syFormat := BYTE#16#07;

	        END_IF;

	    END_REGION

	    REGION Step 17

	        IF #si_StepNr = 17 THEN

	            //Step configuration
	            #sa_Stepconfig.Write := TRUE;
	            #sa_Stepconfig.ParaNo := 11;

	            //Used parameters in this step
	            //p133 - Motor configuration
	            //1 - p133.0 Motor connection type
	            #sa_Parameter[1].siParaNo := 133;
	            #sa_Parameter[1].srValue := #iUDT_MotorConfig.Connection;
	            #sa_Parameter[1].syFormat := BYTE#16#06;
	            //2 - Drive unit line supply voltage
	            #sa_Parameter[2].siParaNo := 210;
	            #sa_Parameter[2].srValue := #iUDT_MotorConfig.MainVoltage;
	            #sa_Parameter[2].syFormat := BYTE#16#06;
	            //3 - Motor type selection
	            #sa_Parameter[3].siParaNo := 300;
	            #sa_Parameter[3].srValue := 1;                              //1: Induction motor
	            #sa_Parameter[3].syFormat := BYTE#16#03;
	            //4 - Rated motor voltage
	            #sa_Parameter[4].siParaNo := 304;
	            #sa_Parameter[4].srValue := #iUDT_MotorConfig.NominalVoltage;
	            #sa_Parameter[4].syFormat := BYTE#16#08;
	            //5 - Rated motor current
	            #sa_Parameter[5].siParaNo := 305;
	            #sa_Parameter[5].srValue := #iUDT_MotorConfig.NominalCurrent;
	            #sa_Parameter[5].syFormat := BYTE#16#08;
	            //6 - Number of motors connected in parallel
	            #sa_Parameter[6].siParaNo := 306;
	            #sa_Parameter[6].srValue := #iUDT_MotorConfig.NoMotorsParallel;
	            #sa_Parameter[6].syFormat := BYTE#16#05;
	            //7 - Rated motor power
	            #sa_Parameter[7].siParaNo := 307;
	            #sa_Parameter[7].srValue := #iUDT_MotorConfig.NominalPower;
	            #sa_Parameter[7].syFormat := BYTE#16#08;
	            //8 - Rated motor power factor
	            #sa_Parameter[8].siParaNo := 308;
	            #sa_Parameter[8].srValue := #iUDT_MotorConfig.CosPhi;
	            #sa_Parameter[8].syFormat := BYTE#16#08;
	            //9 - Rated motor frequency
	            #sa_Parameter[9].siParaNo := 310;
	            #sa_Parameter[9].srValue := 50.0;
	            #sa_Parameter[9].syFormat := BYTE#16#08;
	            //10 - Rated motor speed
	            #sa_Parameter[10].siParaNo := 311;
	            #sa_Parameter[10].srValue := 1450.0;
	            #sa_Parameter[10].syFormat := BYTE#16#08;
	            //11 - Current limit
	            #sa_Parameter[11].siParaNo := 640;
	            #sa_Parameter[11].srValue := #iUDT_MotorConfig.NominalCurrent * 1.5;
	            #sa_Parameter[11].syFormat := BYTE#16#08;

	        END_IF;

	    END_REGION

	    REGION Step 18

	        IF #si_StepNr = 18 THEN

	            //Step configuration
	            #sa_Stepconfig.Read := TRUE;
	            #sa_Stepconfig.Write := TRUE;
	            #sa_Stepconfig.ParaNo := 5;

	            //Used parameters in this step
	            //1 - Ramp-function generator ramp-up time
	            #sa_Parameter[1].siParaNo := 1120;
	            #sa_Parameter[1].srValue := 10.0;
	            #sa_Parameter[1].syFormat := BYTE#16#08;
	            //2 - Ramp-function generator ramp-down time
	            #sa_Parameter[2].siParaNo := 1121;
	            #sa_Parameter[2].srValue := 10.0;
	            #sa_Parameter[2].syFormat := BYTE#16#08;
	            //3 - OFF3 ramp-down time
	            #sa_Parameter[3].siParaNo := 1135;
	            #sa_Parameter[3].srValue := #iUDT_MotorConfig.MinimumRamp;
	            #sa_Parameter[3].syFormat := BYTE#16#08;
	            //4 - Motor holding brake opening time
	            #sa_Parameter[4].siParaNo := 1216;
	            #sa_Parameter[4].srValue := 100.0;
	            #sa_Parameter[4].syFormat := BYTE#16#08;
	            //5 - Motor holding brake closing time
	            #sa_Parameter[5].siParaNo := 1217;
	            #sa_Parameter[5].srValue := 100.0;
	            #sa_Parameter[5].syFormat := BYTE#16#08;

	        END_IF;

	    END_REGION

	    REGION Step 19

	        IF #si_StepNr = 19 THEN

	            //Step configuration
	            #sa_Stepconfig.Read := TRUE;
	            #sa_Stepconfig.Write := TRUE;
	            #sa_Stepconfig.ParaNo := 12;

	            //Used parameters in this step
	            //1 - Reference speed reference frequency
	            #sa_Parameter[1].siParaNo := 2000;
	            #sa_Parameter[1].srValue := 2000.0;
	            #sa_Parameter[1].syFormat := BYTE#16#08;
	            //2 - Reference current
	            #sa_Parameter[2].siParaNo := 2002;
	            #sa_Parameter[2].srValue := #iUDT_MotorConfig.NominalCurrent * 1.5;
	            #sa_Parameter[2].syFormat := BYTE#16#08;
	            //3 - Reference torque
	            #sa_Parameter[3].siParaNo := 2003;
	            #sa_Parameter[3].srValue := #iUDT_MotorConfig.NominalTorque * 1.5;
	            #sa_Parameter[3].syFormat := BYTE#16#08;
	            //4 - Ramp-function generator ramp-up time
	            #sa_Parameter[4].siParaNo := 1120;
	            #sa_Parameter[4].srValue := 20.0;
	            #sa_Parameter[4].syFormat := BYTE#16#08;
	            //5 - Ramp-function generator ramp-down time
	            #sa_Parameter[5].siParaNo := 1121;
	            #sa_Parameter[5].srValue := 20.0;
	            #sa_Parameter[5].syFormat := BYTE#16#08;
	            //Drive commissioning parameter filter
	            //6 - Power unit commissioning
	            #sa_Parameter[6].siParaNo := 10;
	            #sa_Parameter[6].srValue := 2.0;
	            #sa_Parameter[6].syFormat := BYTE#16#03;
	            //7 - Maximum speed
	            #sa_Parameter[7].siParaNo := 1082;
	            #sa_Parameter[7].srValue := 2000.0;
	            #sa_Parameter[7].syFormat := BYTE#16#08;
	            //8 - BI: Jog bit 0
	            #sa_Parameter[8].siParaNo := 1055;
	            #sa_Parameter[8].siIndex := 1;
	            #sa_Parameter[8].syFormat := BYTE#16#07;
	            //9 - BI: Jog bit 1
	            #sa_Parameter[9].siParaNo := 1056;
	            #sa_Parameter[9].siIndex := 1;
	            #sa_Parameter[9].syFormat := BYTE#16#07;
	            //10 - BI: 1st acknowledge faults
	            #sa_Parameter[10].siParaNo := 2103;
	            #sa_Parameter[10].siIndex := 1;
	            #sa_Parameter[10].syFormat := BYTE#16#07;
	            //11 - BI: 2nd acknowledge faults
	            #sa_Parameter[11].siParaNo := 2104;
	            #sa_Parameter[11].syFormat := BYTE#16#07;
	            //12 - BI: Command data set selection CDS bit 0
	            #sa_Parameter[12].siParaNo := 810;
	            #sa_Parameter[12].syFormat := BYTE#16#07;

	        END_IF;

	    END_REGION

	    REGION Step 20

	        IF #si_StepNr = 20 AND #sx_SelectedG120D THEN

	            //Step configuration
	            #sa_Stepconfig.Read := TRUE;
	            #sa_Stepconfig.Write := TRUE;
	            #sa_Stepconfig.ParaNo := 1;

	            //Used parameters in this step
	            //1 - Power unit code number
	            #sa_Parameter[1].siParaNo := 201;
	            #sa_Parameter[1].srValue := #iUDT_MotorConfig.VFDType;
	            #sa_Parameter[1].syFormat := BYTE#16#06;

	        END_IF;

	        IF #si_StepNr = 20 AND #sx_SelectedG120C THEN

	            #si_StepNr := 24;

	        END_IF;

	    END_REGION

	    REGION Step 21

	        IF #si_StepNr = 21 THEN

	            //Step configuration
	            #sa_Stepconfig.Read := TRUE;
	            #sa_Stepconfig.Write := TRUE;
	            #sa_Stepconfig.ParaNo := 1;

	            //Used parameters in this step
	            //1 - Drive commissioning parameter filter
	            #sa_Parameter[1].siParaNo := 10;
	            #sa_Parameter[1].srValue := 4.0;         //4: Encoder commissioning
	            #sa_Parameter[1].syFormat := BYTE#16#03;

	        END_IF;

	    END_REGION

	    REGION Step 22

	        IF #si_StepNr = 22 AND NOT #iUDT_MotorConfig.EncoderConfig THEN

	            //Step configuration
	            #sa_Stepconfig.Read := TRUE;
	            #sa_Stepconfig.Write := TRUE;
	            #sa_Stepconfig.ParaNo := 1;

	            //Used parameters in this step
	            //1 - Encoder type selection
	            #sa_Parameter[1].siParaNo := 400;
	            #sa_Parameter[1].syFormat := BYTE#16#03;

	        END_IF;

	        IF #si_StepNr = 22 AND #iUDT_MotorConfig.EncoderConfig THEN

	            //Step configuration
	            #sa_Stepconfig.Read := TRUE;
	            #sa_Stepconfig.Write := TRUE;
	            #sa_Stepconfig.ParaNo := 4;

	            //Used parameters in this step
	            //1-  Encoder type selection
	            #sa_Parameter[1].siParaNo := 400;
	            #sa_Parameter[1].srValue := 9999.0;         //9999: User-defined
	            #sa_Parameter[1].syFormat := BYTE#16#03;
	            //2 - Rotary encoder pulse number
	            #sa_Parameter[2].siParaNo := 408;
	            #sa_Parameter[2].sdValue := REAL_TO_DINT(#iUDT_MotorConfig.EncoderResolution);
	            #sa_Parameter[2].syFormat := BYTE#16#07;
	            //3 - Encoder rotary zero mark distance
	            #sa_Parameter[3].siParaNo := 425;
	            #sa_Parameter[3].sdValue := REAL_TO_DINT(#iUDT_MotorConfig.EncoderResolution);
	            #sa_Parameter[3].syFormat := BYTE#16#07;
	            //4 - Encoder configuration effective
	            #sa_Parameter[4].siParaNo := 404;
	            #sa_Parameter[4].sdValue := 2097160;
	            #sa_Parameter[4].syFormat := BYTE#16#07;

	        END_IF;

	    END_REGION

	    REGION Step 23

	        IF #si_StepNr = 23 AND #sx_SelectedG120D THEN

	            //Step configuration
	            #sa_Stepconfig.Read := TRUE;
	            #sa_Stepconfig.Write := TRUE;
	            #sa_Stepconfig.ParaNo := 2;

	            //Used parameters in this step
	            //1 - Open-loop/closed-loop control operating mode
	            IF #iUDT_MotorConfig.EncoderConfig THEN
	                #sa_Parameter[1].siParaNo := 1300;
	                #sa_Parameter[1].srValue := 21.0;           //21: Speed control (with encoder)
	                #sa_Parameter[1].syFormat := BYTE#16#03;

	            ELSE
	                //1 - Open-loop/closed-loop control operating mode
	                #sa_Parameter[1].siParaNo := 1300;
	                #sa_Parameter[1].srValue := 20.0;           //20 - Speed control (encoderless)
	                #sa_Parameter[1].syFormat := BYTE#16#03;

	            END_IF;

	            //2 - Drive commissioning parameter filter
	            #sa_Parameter[2].siParaNo := 10;
	            #sa_Parameter[2].srValue := 1.0;                //1: Quick commissioning
	            #sa_Parameter[2].syFormat := BYTE#16#03;

	        END_IF;

	    END_REGION

	    REGION Step 24

	        IF #si_StepNr = 24 THEN

	            //Step configuration
	            #sa_Stepconfig.Write := TRUE;
	            #sa_Stepconfig.ParaNo := 1;

	            //Used parameters in this step
	            //1 - Save parameters
	            #sa_Parameter[1].siParaNo := 971;
	            #sa_Parameter[1].srValue := 1.0;
	            #sa_Parameter[1].syFormat := BYTE#16#06;

	        END_IF;

	    END_REGION

	    REGION Step 25

	        IF #si_StepNr = 25 THEN

	            //Step configuration
	            #sa_Stepconfig.Read := TRUE;
	            #sa_Stepconfig.ParaNo := 1;

	            //Used parameters in this step
	            //1 - Save parameters
	            #sa_Parameter[1].siParaNo := 971;
	            #sa_Parameter[1].syFormat := BYTE#16#06;

	        END_IF;

	    END_REGION

	    REGION Step 26

	        IF #si_StepNr = 26 THEN

	            //Step configuration
	            #sa_Stepconfig.Read := TRUE;
	            #sa_Stepconfig.Write := TRUE;
	            #sa_Stepconfig.ParaNo := 1;

	            //Used parameters in this step
	            //1 - Drive commissioning parameter filter
	            #sa_Parameter[1].siParaNo := 10;
	            #sa_Parameter[1].syFormat := BYTE#16#03;

	        END_IF;

	    END_REGION

	    REGION Step 27

	        IF #si_StepNr = 27 THEN

	            //Step configuration
	            #sa_Stepconfig.Read := TRUE;
	            #sa_Stepconfig.Write := TRUE;
	            #sa_Stepconfig.ParaNo := 1;

	            //Used parameters in this step
	            //1 - Drive commissioning parameter filter
	            #sa_Parameter[1].siParaNo := 10;
	            #sa_Parameter[1].srValue := 95.0;           //95 - Safety Integrated commissioning
	            #sa_Parameter[1].syFormat := BYTE#16#03;

	        END_IF;

	    END_REGION

	    REGION Step 28

	        IF #si_StepNr = 28 THEN

	            //Step configuration
	            #sa_Stepconfig.Write := TRUE;
	            #sa_Stepconfig.ParaNo := 3;

	            //Used parameters in this step
	            //1 - SI password input
	            #sa_Parameter[1].siParaNo := 9761;
	            #sa_Parameter[1].syFormat := BYTE#16#07;
	            //2 - SI password new
	            #sa_Parameter[2].siParaNo := 9762;
	            #sa_Parameter[2].syFormat := BYTE#16#07;
	            //3 - SI password acknowledgment
	            #sa_Parameter[3].siParaNo := 9763;
	            #sa_Parameter[3].syFormat := BYTE#16#07;

	        END_IF;

	    END_REGION

	    REGION Step 29

	        IF #si_StepNr = 29 THEN

	            //Step configuration
	            #sa_Stepconfig.Write := TRUE;
	            #sa_Stepconfig.ParaNo := 1;

	            //Used parameters in this step
	            //1 - SI password input
	            #sa_Parameter[1].siParaNo := 9761;
	            #sa_Parameter[1].syFormat := BYTE#16#07;

	        END_IF;

	    END_REGION

	    REGION Step 30

	        IF #si_StepNr = 30 THEN

	            //Step configuration
	            #sa_Stepconfig.Read := TRUE;
	            #sa_Stepconfig.Write := TRUE;
	            #sa_Stepconfig.ParaNo := 4;

	            //Used parameters in this step 1
	            //1 - SI enable functions integrated in the drive
	            #sa_Parameter[1].siParaNo := 9601;
	            #sa_Parameter[1].sdValue := 8;
	            #sa_Parameter[1].syFormat := BYTE#16#07;
	            //2 - SI PROFIsafe address
	            #sa_Parameter[2].siParaNo := 9610;
	            #sa_Parameter[2].srValue := #iUDT_MotorConfig.FAdress;
	            #sa_Parameter[2].syFormat := BYTE#16#06;
	            //3 - PROFIsafe telegram selection
	            #sa_Parameter[3].siParaNo := 60022;
	            #sa_Parameter[3].srValue := 30.0;
	            #sa_Parameter[3].syFormat := BYTE#16#06;
	            //4 - SI forced checking procedure timer
	            #sa_Parameter[4].siParaNo := 9659;
	            #sa_Parameter[4].srValue := 9000.0;
	            #sa_Parameter[4].syFormat := BYTE#16#08;

	        END_IF;

	    END_REGION

	    REGION Step 31

	        IF #si_StepNr = 31 THEN

	            //Step configuration
	            #sa_Stepconfig.Write := TRUE;
	            #sa_Stepconfig.ParaNo := 1;

	            //Used parameters in this step
	            //1 - SI Motion copy function
	            #sa_Parameter[1].siParaNo := 9700;
	            #sa_Parameter[1].srValue := 208.0;
	            #sa_Parameter[1].syFormat := BYTE#16#03;

	        END_IF;

	    END_REGION

	    REGION Step 32

	        IF #si_StepNr = 32 THEN

	            //Step configuration
	            #sa_Stepconfig.Read := TRUE;
	            #sa_Stepconfig.ParaNo := 1;

	            //Used parameters in this step
	            //1 - SI Motion copy function
	            #sa_Parameter[1].siParaNo := 9700;
	            #sa_Parameter[1].syFormat := BYTE#16#03;

	        END_IF;

	    END_REGION

	    REGION Step 33

	        IF #si_StepNr = 33 THEN

	            //Step configuration
	            #sa_Stepconfig.Read := TRUE;
	            #sa_Stepconfig.ParaNo := 2;

	            //Used parameters in this step
	            //1 - SI enable functions integrated in the drive
	            #sa_Parameter[1].siParaNo := 9801;
	            #sa_Parameter[1].srValue := 8.0;
	            #sa_Parameter[1].syFormat := BYTE#16#06;
	            //2 - Safety adress
	            #sa_Parameter[2].siParaNo := 9810;
	            #sa_Parameter[2].srValue := #iUDT_MotorConfig.FAdress;
	            #sa_Parameter[2].syFormat := BYTE#16#06;

	        END_IF;

	    END_REGION

	    REGION Step 34

	        IF #si_StepNr = 34 THEN

	            //Step configuration
	            #sa_Stepconfig.Write := TRUE;
	            #sa_Stepconfig.ParaNo := 1;

	            //Used parameters in this step
	            //1 - Acknowledge SI data change
	            #sa_Parameter[1].siParaNo := 9701;
	            #sa_Parameter[1].srValue := 220.0;          //220: [DC hex] Acknowledge SI basic parameter change
	            #sa_Parameter[1].syFormat := BYTE#16#03;

	        END_IF;

	    END_REGION

	    REGION Step 35

	        IF #si_StepNr = 35 THEN

	            //Step configuration
	            #sa_Stepconfig.Read := TRUE;
	            #sa_Stepconfig.ParaNo := 1;

	            //Used parameters in this step
	            //1 - Acknowledge SI data change
	            #sa_Parameter[1].siParaNo := 9701;
	            #sa_Parameter[1].syFormat := BYTE#16#03;

	        END_IF;

	    END_REGION

	    REGION Step 36

	        IF #si_StepNr = 36 THEN

	            //Step configuration
	            #sa_Stepconfig.Write := TRUE;
	            #sa_Stepconfig.ParaNo := 1;

	            //Used parameters in this step
	            //1 - SI copy function
	            #sa_Parameter[1].siParaNo := 9700;
	            #sa_Parameter[1].srValue := 87.0;           //87: [57 hex] Start copy function SI parameters
	            #sa_Parameter[1].syFormat := BYTE#16#03;

	        END_IF;

	    END_REGION

	    REGION Step 37

	        IF #si_StepNr = 37 THEN

	            //Step configuration
	            #sa_Stepconfig.Read := TRUE;
	            #sa_Stepconfig.ParaNo := 1;

	            //Used parameters in this step
	            //1 - SI copy function
	            #sa_Parameter[1].siParaNo := 9700;
	            #sa_Parameter[1].syFormat := BYTE#16#03;


	        END_IF;

	    END_REGION

	    REGION Step 38

	        IF #si_StepNr = 38 THEN

	            //Step configuration
	            #sa_Stepconfig.Write := TRUE;
	            #sa_Stepconfig.ParaNo := 1;

	            //Used parameters in this step
	            //1 - Acknowledge SI data change
	            #sa_Parameter[1].siParaNo := 9701;
	            #sa_Parameter[1].srValue := 220.0;          //220: [DC hex] Acknowledge SI basic parameter change
	            #sa_Parameter[1].syFormat := BYTE#16#03;

	        END_IF;

	    END_REGION

	    REGION Step 39

	        IF #si_StepNr = 39 THEN

	            //Step configuration
	            #sa_Stepconfig.Read := TRUE;
	            #sa_Stepconfig.ParaNo := 1;

	            //Used parameters in this step
	            //1 - Acknowledge SI data change
	            #sa_Parameter[1].siParaNo := 9701;
	            #sa_Parameter[1].syFormat := BYTE#16#03;

	        END_IF;

	    END_REGION

	    REGION Step 40

	        IF #si_StepNr = 40 THEN

	            //Step configuration
	            #sa_Stepconfig.Read := TRUE;
	            #sa_Stepconfig.Write := TRUE;
	            #sa_Stepconfig.ParaNo := 1;

	            //1 - Drive commissioning parameter filter
	            #sa_Parameter[1].siParaNo := 10;
	            #sa_Parameter[1].syFormat := 3;

	        END_IF;

	    END_REGION

	    REGION Step 41

	        IF #si_StepNr = 41 THEN

	            //Step configuration
	            #sa_Stepconfig.Write := TRUE;
	            #sa_Stepconfig.ParaNo := 1;

	            //Used parameters in this step
	            //1 - Save parameters
	            #sa_Parameter[1].siParaNo := 971;
	            #sa_Parameter[1].srValue := 1.0;            //1: Save drive object
	            #sa_Parameter[1].syFormat := BYTE#16#06;

	        END_IF;

	    END_REGION

	    REGION Step 42

	        IF #si_StepNr = 42 THEN

	            //Step configuration
	            #sa_Stepconfig.Read := TRUE;
	            #sa_Stepconfig.ParaNo := 2;

	            //Used parameters in this step
	            //1 - Reset drive parameters
	            #sa_Parameter[1].siParaNo := 970;
	            #sa_Parameter[1].syFormat := BYTE#16#06;
	            //2 - Parameter write inhibit status
	            #sa_Parameter[2].siParaNo := 3996;
	            #sa_Parameter[2].syFormat := BYTE#16#05;

	        END_IF;

	    END_REGION

	    REGION Step 43

	        IF #si_StepNr = 43 THEN

	            //Step configuration
	            #sa_Stepconfig.Write := TRUE;
	            #sa_Stepconfig.ParaNo := 1;

	            //Used parameters in this step
	            //1 - Drive unit reset
	            #sa_Parameter[1].siParaNo := 972;
	            #sa_Parameter[1].srValue := 1.0;            //1: Hardware-Reset immediate
	            #sa_Parameter[1].syFormat := 16#0006;
	            #sa_Parameter[1].swErrorNo := 0;

	            #sa_Status.NeedAck := TRUE;

	        END_IF;

	    END_REGION

	    REGION Step 44

	        IF #si_StepNr = 44 THEN

	            //Step configuration
	            #sa_Stepconfig.Read := TRUE;
	            #sa_Stepconfig.ParaNo := 1;

	            //Used parameters in this step
	            //1 - Drive commissioning parameter filter
	            #sa_Parameter[1].siParaNo := 10;
	            #sa_Parameter[1].syFormat := 16#0003;
	            #sa_Parameter[1].swErrorNo := 0;

	        END_IF;

	    END_REGION

	    REGION Step 45

	        IF #si_StepNr = 45 THEN

	            //Step configuration
	            #sa_Stepconfig.Read := TRUE;
	            #sa_Stepconfig.Write := TRUE;
	            #sa_Stepconfig.ParaNo := 1;

	            //Used parameters in this step
	            //1 - Drive commissioning parameter filter
	            #sa_Parameter[1].siParaNo := 10;
	            #sa_Parameter[1].syFormat := BYTE#16#03;
	            #sa_Parameter[1].swErrorNo := 0;

	        END_IF;

	    END_REGION

	    REGION Step 46

	        IF #si_StepNr = 46 THEN

	            //Step configuration
	            #sa_Stepconfig.Read := TRUE;
	            #sa_Stepconfig.Write := TRUE;
	            #sa_Stepconfig.ParaNo := 2;

	            //Used parameters in this step
	            //1 - Temperature sensor, sensor type
	            #sa_Parameter[1].siParaNo := 601;
	            #sa_Parameter[1].srValue := #iUDT_MotorConfig.ThermalConfig;
	            #sa_Parameter[1].syFormat := BYTE#16#03;

	            //2 - Motor holding brake configuration
	            #sa_Parameter[2].siParaNo := 1215;
	            #sa_Parameter[2].srValue := 0;
	            #sa_Parameter[2].syFormat := BYTE#16#03;

	            IF #iUDT_MotorConfig.BrakeConfig THEN

	                IF #sx_SelectedG120C THEN

	                    #sa_Parameter[2].srValue := 3;

	                END_IF;

	                IF #sx_SelectedG120D THEN

	                    #sa_Parameter[2].srValue := 1;

	                END_IF;

	            END_IF;

	        END_IF;

	    END_REGION

	    REGION Step 47

	        IF #si_StepNr = 47 THEN

	            //Step configuration
	            #sa_Stepconfig.Read := TRUE;
	            #sa_Stepconfig.Write := TRUE;
	            #sa_Stepconfig.ParaNo := 1;

	            //Used parameters in this step
	            //1 - Motor data identification and rotating measurement
	            #sa_Parameter[1].siParaNo := 1900;
	            #sa_Parameter[1].srValue := 2.0;            //2: Identifying motor data (at standstill)
	            #sa_Parameter[1].syFormat := BYTE#16#03;

	        END_IF;

	    END_REGION

	    REGION Step 48

	        IF #si_StepNr = 48 AND #sx_SelectedG120D THEN

	            //Step configuration
	            #sa_Stepconfig.Read := TRUE;
	            #sa_Stepconfig.ParaNo := 2;

	            //Used parameters in this step
	            //1 - Identification status
	            #sa_Parameter[1].siParaNo := 47;
	            #sa_Parameter[1].syFormat := BYTE#16#03;
	            //2 - Motor data identification and rotating measurement
	            #sa_Parameter[2].siParaNo := 1900;
	            #sa_Parameter[2].syFormat := BYTE#16#03;

	            #sx_StartMeasuring := TRUE;

	        END_IF;

	        IF #si_StepNr = 48 AND #sx_SelectedG120C THEN

	            //Step configuration
	            #sa_Stepconfig.Read := TRUE;
	            #sa_Stepconfig.ParaNo := 2;

	            //1 - Used parameters in this step
	            //Identification status
	            #sa_Parameter[1].siParaNo := 47;
	            #sa_Parameter[1].syFormat := BYTE#16#03;
	            //2 - Motor data identification and rotating measurement
	            #sa_Parameter[2].siParaNo := 1900;
	            #sa_Parameter[2].syFormat := BYTE#16#03;
	            //3 - Status word 1
	            #sa_Parameter[3].siParaNo := 52;
	            #sa_Parameter[3].srValue := 60272.0;
	            #sa_Parameter[3].syFormat := BYTE#16#06;

	            #sx_StartMeasuring := TRUE;

	        END_IF;

	    END_REGION

	    REGION Step 49

	        IF #si_StepNr = 49 THEN

	            //Step configuration
	            #sa_Stepconfig.Write := TRUE;
	            #sa_Stepconfig.Read := TRUE;
	            #sa_Stepconfig.ParaNo := 1;

	            //Used parameters in this step
	            //1 - Save parameters
	            #sa_Parameter[1].siParaNo := 971;
	            #sa_Parameter[1].srValue := 1.0;            //1: Save drive object
	            #sa_Parameter[1].syFormat := BYTE#16#06;

	        END_IF;

	    END_REGION

	    REGION Step 50

	        IF #si_StepNr = 50 THEN

	            //Step configuration
	            #sa_Stepconfig.Read := TRUE;
	            #sa_Stepconfig.ParaNo := 1;

	            //Used parameters in this step
	            //1 - Save parameters
	            #sa_Parameter[1].siParaNo := 971;
	            #sa_Parameter[1].syFormat := BYTE#16#06;

	        END_IF;

	    END_REGION

	    REGION Step 51

	        IF #si_StepNr = 51 THEN

	            //Step configuration
	            #sa_Stepconfig.Read := TRUE;
	            #sa_Stepconfig.ParaNo := 1;

	            //Used parameters in this step
	            //1 - Memory card status
	            #sa_Parameter[1].siParaNo := 9400;
	            #sa_Parameter[1].syFormat := BYTE#16#03;

	        END_IF;

	    END_REGION

	    REGION Step 52

	        IF #si_StepNr = 52 THEN


	            IF #sa_Status.MemoryCardInserted THEN

	                //Step configuration
	                #sa_Stepconfig.Write := TRUE;
	                #sa_Stepconfig.ParaNo := 1;

	                //Used parameters in this step
	                //1 - Data transfer start
	                #sa_Parameter[1].siParaNo := 804;
	                #sa_Parameter[1].srValue := 2.0;            //2:start data transfer from device memory to memory card
	                #sa_Parameter[1].syFormat := BYTE#16#03;

	            ELSE

	                #si_StepNr := 54;

	            END_IF;

	        END_IF;

	    END_REGION

	    REGION Step 53

	        IF #si_StepNr = 53 THEN

	            //Step configuration
	            #sa_Stepconfig.Read := TRUE;
	            #sa_Stepconfig.ParaNo := 1;

	            //Used parameters in this step
	            //1 - Data transfer start
	            #sa_Parameter[1].siParaNo := 804;
	            #sa_Parameter[1].srValue := 0.0;
	            #sa_Parameter[1].syFormat := BYTE#16#03;

	        END_IF;

	    END_REGION

	    REGION Step 54

	        IF #si_StepNr = 54 THEN

	            //Step configuration
	            #sa_Stepconfig.Read := TRUE;
	            #sa_Stepconfig.Write := TRUE;
	            #sa_Stepconfig.ParaNo := 1;

	            //Used parameters in this step
	            //1 - Drive commissioning parameter filter
	            #sa_Parameter[1].siParaNo := 10;
	            #sa_Parameter[1].syFormat := BYTE#16#03;

	            #sx_Done := TRUE;
	            #sx_Busy := FALSE;
	            #sx_StartMeasuring := FALSE;

	        END_IF;

	    END_REGION

	END_REGION

	REGION 5 - Prepered data

	    //This region is responsible for preparing data for each step. Copying data from the sequence and activating the write / read mode or both.
	    IF (#sx_Start AND                   // If occurs: signal to start of parametrization
	        NOT #sx_PreparedData AND        // And step data is not prepared
	        NOT #sx_Done AND                // And parametrization is not done
	        #ix_Enable)                     // And input enable signal
	    THEN

	        REGION 5.1 - Parametrization mode - only read

	            //Set READ mode
	            IF (#sa_Stepconfig.Read
	                AND NOT #sa_Stepconfig.Write)
	            THEN

	                #sx_OnlyRead := TRUE;
	                #sx_OnlyWrite := FALSE;
	                #sx_WriteRead := FALSE;
	                #sx_SinaParaStart := TRUE;
	                #sx_SinaParaReadWrite := FALSE;

	            END_IF;

	        END_REGION

	        REGION 5.2 - Parametrization mode - only write

	            //Set WRITE mode
	            IF (NOT #sa_Stepconfig.Read
	                AND #sa_Stepconfig.Write)
	            THEN

	                #sx_OnlyRead := FALSE;
	                #sx_OnlyWrite := TRUE;
	                #sx_WriteRead := FALSE;
	                #sx_SinaParaStart := TRUE;
	                #sx_SinaParaReadWrite := TRUE;

	            END_IF;

	        END_REGION

	        REGION 5.3 - Parametrization mode - write and read

	            //Set READ/WRITE mode
	            IF (#sa_Stepconfig.Read
	                AND #sa_Stepconfig.Write)
	            THEN

	                #sx_OnlyRead := FALSE;
	                #sx_OnlyWrite := FALSE;
	                #sx_WriteRead := TRUE;
	                #sx_SinaParaStart := TRUE;
	                #sx_SinaParaReadWrite := TRUE;

	            END_IF;

	        END_REGION

	        #si_SinaParaParaNo := #sa_Stepconfig.ParaNo;          // Copy number of parameters from step commissionig to static number of parameters
	        #sa_ParameterToCompare := #sa_Parameter;               // Copy parameters
	        #sx_PreparedData := TRUE;                              // Set step data prepared

	    END_IF;

	END_REGION

	REGION 6 - Call read/write parameter block - SinaPara

	    // Sina Para is responsible for write and reads parameters from VFD
	    #sFB_SinaParaInstance(Start := #sx_SinaParaStart
	                          AND #sx_Start
	                          AND #ix_Enable,
	                          ReadWrite := #sx_SinaParaReadWrite,
	                          ParaNo := #si_SinaParaParaNo,
	                          AxisNo := #cb_SinaParamAxisNo,
	                          hardwareId := #ihw_SinaParamHardwareId,
	                          Ready => #sx_SinaParaReady,
	                          Busy => #sx_SinaParaBusy,
	                          Done => #sx_SinaParaDone,
	                          Error => #sa_SinaPara.Error,
	                          ErrorId => #sa_SinaPara.ErrorId,
	                          DiagId => #sa_SinaPara.DiagId,
	                          Parameter := #sa_Parameter);

	END_REGION

	REGION 7 - Compare read parameters with basic parameters

	    // When the comparison parameters have incorrect value or format, function SinaPara reads again parameters
	    IF (#sx_ResponseValueError OR
	        #sx_WrongFormat)
	    THEN

	        #sx_SinaParaStart := TRUE;
	        #sx_SinaParaDone := FALSE;
	        #sx_ResponseValueError := FALSE;
	        #sx_WrongFormat := FALSE;

	    END_IF;

	    // After read correctly data with SinaPara are compered with the parameter from this step.
	    IF (#sx_SinaParaStart AND                                                                                                                           // If SinaPara start signal is on
	        NOT #sx_SinaParaReadWrite AND                                                                                                                   // And SinaPara is read parameters
	        #sx_SinaParaDone AND                                                                                                                            // And SinaPara function is done is on
	        NOT #sa_SinaPara.Error AND                                                                                                                      // And SinaPara function error signal is off
	        #ix_Enable)                                                                                                                                     // And input enable signal
	    THEN

	        // Create loop from 1 parameter to number of parameters
	        FOR #si_Loop := 1 TO #si_SinaParaParaNo DO

	            // If parameter value from data of parameters are different than parameter value from step commissioning
	            IF
	                #sa_Parameter[#si_Loop].srValue <> #sa_ParameterToCompare[#si_Loop].srValue OR
	                #sa_Parameter[#si_Loop].sdValue <> #sa_ParameterToCompare[#si_Loop].sdValue
	            THEN

	                #sx_ResponseValueError := TRUE;
	                #si_ParameterNrError := #si_Loop;
	                #si_StepNrError := #si_StepNr;

	            ELSE

	                #sx_ResponseValueError := False;

	            END_IF;

	            // If parameter format is equal 44 set wrong format fault
	            IF #sa_Parameter[#si_Loop].syFormat = 44
	            THEN

	                #sx_WrongFormat := TRUE;
	                #si_ParameterNrError := #si_Loop;
	                #si_StepNrError := #si_StepNr;

	            ELSE

	                #sx_WrongFormat := False;

	            END_IF;

	        END_FOR;

	        // Check if error occurs if isn't then read parameter are the same like step parameters. Else the SinaPara read parameters again.
	        IF (NOT #sx_ResponseValueError AND
	            NOT #sx_WrongFormat) OR
	            #si_StepNr = 51
	        THEN

	            #sx_ComparisonParameters := TRUE;

	        ELSE

	            #sx_SinaParaStart := FALSE;

	        END_IF;

	    END_IF;

	    REGION 7.1 - Check if SD is inside

	        IF (#si_StepNr = 51 AND #sa_Parameter[1].srValue = 1) THEN

	            #sa_Status.MemoryCardInserted := TRUE;

	        END_IF;

	    END_REGION

	END_REGION

	REGION 8 - Status commissioning

	    REGION 8.1 - Step number Error

	        IF (#sx_SinaParaStart AND                                                                   // Parametrization is start
	            #sa_SinaPara.Error AND                                                                  // Occurs error bit
	            (NOT #sa_Status.NeedAck) AND                                                            // This step does not need to be confirmed
	            (NOT #sx_SinaParaReadWrite OR                                                           // Parameters are not write
	            (#sx_SinaParaReadWrite AND                                                              // Parameters are read
	            #sx_ReadTime)))                                                                         // Read time signal is on
	        THEN

	            #sa_Status.StepNrError := #si_StepNr;
	            #sx_Start := FALSE;
	            #sx_Error := TRUE;
	            #sx_Done := FALSE;
	            #sx_StartMeasuring := FALSE;

	        END_IF;

	        IF #sa_Status.NeedAck AND                                                       // This step must be confirmed
	            #sa_SinaPara.Error                                                          // Occurs error bit

	        THEN

	            #sx_SinaParaStart := FALSE;

	        END_IF;

	    END_REGION

	    REGION 8.2 - Read Done

	        // The parameters are read form VFD
	        IF (#sx_SinaParaStart                       // Parametrization is start
	            AND #sx_SinaParaDone                    // Parametrization is done
	            AND NOT #sx_SinaParaReadWrite AND       // Parameters are not read/write
	            (#sx_OnlyRead OR #sx_WriteRead) AND     // Is selected only read mode or is selected wite/read mode
	            #sx_ComparisonParameters AND            // Comparison parameters are correct
	            #ix_Enable)
	        THEN

	            #sx_ReadDone := TRUE;                   // Set read done
	            #sx_SinaParaStart := FALSE;             // Stop parametrization

	        END_IF;

	    END_REGION

	    REGION 8.3 - Write Done

	        // The parameters are write to VFD
	        IF (#sx_SinaParaStart                             // Parametrization is start
	            AND #sx_SinaParaDone                          // Parametrization is done
	            AND #sx_SinaParaReadWrite                     // Parameters are write signal is on
	            AND (#sx_OnlyWrite OR #sx_WriteRead)          // Is selected only write mode or is selected wite/read mode
	            AND #ix_Enable)
	        THEN

	            #sx_WriteDone := TRUE;
	            #sx_SinaParaStart := FALSE;
	            #sx_SinaParaReadWrite := FALSE;
	            #sx_SinaParaDone := FALSE;
	            #sx_StartDelayTime := TRUE;

	        END_IF;

	        // Write parameters in VFD need 1 sec to read
	        IF #sx_StartDelayTime
	        THEN

	            // Monitor rising trigger if occur system clock bit 1Hz
	            #sR_TRIG_DelayTime(CLK := "DB_Memory"."Clock_0.5Hz");

	            // If trigger for time couting occurs then increase step time by 1 [s]
	            IF #sR_TRIG_DelayTime.Q
	            THEN

	                #si_DelayTime += 1;

	            END_IF;

	            // If the deley time is bigger as 2
	            IF #si_DelayTime >= 2
	            THEN

	                #si_DelayTime := 0;
	                #sx_StartDelayTime := FALSE;
	                #sx_SinaParaStart := TRUE;

	            END_IF;

	        END_IF;

	    END_REGION

	END_REGION

	REGION 9 - Read Data

	    // Parameter are raed in the loop. At this time the parameters are comparable to those of the step. If they disagree an error occurs
	    IF (((#sx_WriteRead AND #sx_WriteDone)                                         // Write/read mode is selected and write is done
	        OR #sx_OnlyRead)                                                           // Only read mode is selected
	        AND #sx_PreparedData                                                       // Data are prepared
	        AND NOT #sx_Error                                                          // Not error occurs
	        AND NOT #sa_Status.TimeExceeded                                            // Not time step exceeded
	        AND NOT #sx_ReadDone                                                       // Read is not done
	        AND #ix_Enable)                                                            // Input enable signal
	    THEN

	        // Monitor rising trigger if occur system clock bit 1Hz
	        #sR_TRIG_Time(CLK := "DB_Memory".Clock_1Hz);

	        // Increase step time by 1 [s]
	        IF #sR_TRIG_Time.Q                                                            // If trigger for time couting occurs
	        THEN

	            #si_StepTime += 1;

	        END_IF;

	        // If step time is greater than or equal to
	        IF #si_StepTime >= #ci_StepTime
	        THEN

	            #sx_ReadTime := FALSE;


	            IF NOT #sx_ReadDone THEN

	                #sx_Error := TRUE;
	                #sa_Status.TimeExceeded := true;
	                #sa_Status.ResponseValueError := #sx_ResponseValueError;
	                #sa_Status.WrongFormat := #sx_WrongFormat;
	                #sa_Status.StepNrError := #si_StepNrError;
	                #sa_Status.ParameterNrError := #si_ParameterNrError;

	            END_IF;

	        ELSE

	            #sx_ReadTime := TRUE;           // Reset read time

	        END_IF;

	    ELSE

	        #si_StepTime := 0;          // Set step time to 0

	    END_IF;

	END_REGION

	REGION 10 - Freecycle

	    //SinaPara block needs a positive edge to start working
	    IF #sa_Status.StepDone      // If step is done
	        AND #ix_Enable         // Enagle signal is active
	    THEN

	        #sx_Freecycle := TRUE;

	    END_IF;

	END_REGION

	REGION 11 - Step Done

	    // When the step modes are fulfilled, the step done signal is active
	    IF (#sx_ReadDone                          // Read is done
	        AND #sx_WriteDone                     // Write is done
	        AND #sx_WriteRead                     // Write/Read mode is selected
	        AND #sx_ComparisonParameters)         // Comparison read data is done

	        OR (NOT #sx_ReadDone                  // Read isn't done
	        AND #sx_WriteDone                     // Write is done
	        AND #sx_OnlyWrite)                    // Write mode is selected

	        OR (#sx_ReadDone                      // Read is done
	        AND NOT #sx_WriteDone                 // Write isn't done
	        AND #sx_OnlyRead                      // Read mode is selected
	        AND #sx_ComparisonParameters)         // Comparison read data is done
	        AND #ix_Enable                        // Enable signal is active
	    THEN

	        #sa_Status.StepDone := TRUE;

	    END_IF;

	END_REGION

	REGION 12 - Go to next step

	    // When all conditions are met the functions go to the next step automatically or is active signal wich every steps must be acknowledged
	    IF (((#sx_ActiveButtonGoToNextStep                                            // Activeted button to go for the next step
	        AND #iqx_GoToNextStep)                                                    // Signal go to next step is occurs
	        OR NOT #sx_ActiveButtonGoToNextStep)                                      // Signal go to next step is not occurs
	        AND ((#sa_Status.NeedAck                                                  // Need acknowledge
	        AND #iqx_GoToNextStep)                                                    // Activeted button to go for the next step
	        OR NOT #sa_Status.NeedAck)                                                // Need acknowledge is not occurs
	        AND ((NOT #sx_Error                                                       // Is no error
	        AND #sa_Status.StepDone                                                   // Step is done
	        AND #sx_Freecycle)                                                        // Empty cycle
	        OR #sa_Status.NeedAck)                                                    // This step must be confirmed
	        AND #ix_Enable)                                                           // Input enable signal

	    THEN

	        #sx_PreparedData := FALSE;
	        #sx_ReadDone := FALSE;
	        #sx_WriteDone := FALSE;
	        #sx_SinaParaStart := FALSE;
	        #sx_Freecycle := FALSE;
	        #sx_StartMeasuring := FALSE;
	        #sx_ComparisonParameters := FALSE;
	        #iqx_GoToNextStep := FALSE;
	        #sa_Status.NeedAck := FALSE;
	        #sa_Status.StepDone := FALSE;
	        #si_StepNr += 1;

	    END_IF;

	END_REGION

	REGION 13 - Write output

	    #sa_Status.StepNr := #si_StepNr;
	    #qx_Busy := #sx_Busy;
	    #qx_Done := #sx_Done;
	    #qx_Error := #sx_Error;
	    #qx_StartMeasuring := #sx_StartMeasuring;

	END_REGION
END_FUNCTION_BLOCK

TYPE "UDT_VfdSEWSpeedPI"
TITLE = UDT_VFD_SEW_PI
VERSION : 0.1
//User-defined structure of VFD SEW input telegram.
   STRUCT
      Status_Word_1 : Struct   // Status Word 1
         Error { ExternalAccessible := 'False'; ExternalVisible := 'False'; ExternalWritable := 'False'} : Bool;   // An error is active "1"
         Warning { ExternalAccessible := 'False'; ExternalVisible := 'False'; ExternalWritable := 'False'} : Bool;   // A warning is active "1"
         DriveTrain2Active { ExternalAccessible := 'False'; ExternalVisible := 'False'; ExternalWritable := 'False'} : Bool;   // Drive train 2 is active "1"
         VelocityTargetActualComparison { ExternalAccessible := 'False'; ExternalVisible := 'False'; ExternalWritable := 'False'} : Bool;   // The notification "Velocity target-actual-comparison" is on "1"
         SW_LimitSwitchInactive { ExternalAccessible := 'False'; ExternalVisible := 'False'; ExternalWritable := 'False'} : Bool;   // he software limit switch is inactive "1"
         BIT_13_Reserved { ExternalAccessible := 'False'; ExternalVisible := 'False'; ExternalWritable := 'False'} : Bool;   // Reserved
         StandbyActive { ExternalAccessible := 'False'; ExternalVisible := 'False'; ExternalWritable := 'False'} : Bool;   // Standby mode is active "1"
         MovikitHandshakeOut { ExternalAccessible := 'False'; ExternalVisible := 'False'; ExternalWritable := 'False'} : Bool;   // Copied value of "MovikitHandshakeIn"
         InverterReady { ExternalAccessible := 'False'; ExternalVisible := 'False'; ExternalWritable := 'False'} : Bool;   // There's no error and the inverter is ready "1"
         STO_Inactive { ExternalAccessible := 'False'; ExternalVisible := 'False'; ExternalWritable := 'False'} : Bool;   // STO is not active "1"
         OutputStageEnabled { ExternalAccessible := 'False'; ExternalVisible := 'False'; ExternalWritable := 'False'} : Bool;   // The output stage is released "1"
         BrakeReleased { ExternalAccessible := 'False'; ExternalVisible := 'False'; ExternalWritable := 'False'} : Bool;   // The brake is released "1"
         DriveActive { ExternalAccessible := 'False'; ExternalVisible := 'False'; ExternalWritable := 'False'} : Bool;   // The drive is active and the shaft turning "1"
         Referenced { ExternalAccessible := 'False'; ExternalVisible := 'False'; ExternalWritable := 'False'} : Bool;   // The drive is referenced "1"
         RelativePositionApplied { ExternalAccessible := 'False'; ExternalVisible := 'False'; ExternalWritable := 'False'} : Bool;   // The relative position is applied "1"
         InPosition { ExternalAccessible := 'False'; ExternalVisible := 'False'; ExternalWritable := 'False'} : Bool;   // The notification "in position" is on "1"
      END_STRUCT;
      ActualSpeed : Int;   // Actual drive speed (Int) in rpm
      StatusErrorNo : Word;   // Current status of the drive
      ActualTorque : Int;   // Actual torque in percent od the rated unit torque
   END_STRUCT;

END_TYPE

TYPE "UDT_VfdSEWSpeedPO"
TITLE = UDT_VFD_SEW_PO
VERSION : 0.1
//User-defined structure of VFD SEW output telegram.
   STRUCT
      Control_Word_1 : Struct   // Control Word 1
         ResetError { ExternalAccessible := 'False'; ExternalVisible := 'False'; ExternalWritable := 'False'} : Bool;   // Reset error "1"
         BIT_09_Reserved { ExternalAccessible := 'False'; ExternalVisible := 'False'; ExternalWritable := 'False'} : Bool;   // Reserved
         ActivateDriveTrain2 { ExternalAccessible := 'False'; ExternalVisible := 'False'; ExternalWritable := 'False'} : Bool;   // Activate drive train 2 "1"
         BIT_11_Reserved { ExternalAccessible := 'False'; ExternalVisible := 'False'; ExternalWritable := 'False'} : Bool;   // Reserved
         DeactivateSW_LimitSwitch { ExternalAccessible := 'False'; ExternalVisible := 'False'; ExternalWritable := 'False'} : Bool;   // Deactivate software limit switch "1"
         ActivateInhibit { ExternalAccessible := 'False'; ExternalVisible := 'False'; ExternalWritable := 'False'} : Bool;   // Activate inhibit "1"
         ActivateStandby { ExternalAccessible := 'False'; ExternalVisible := 'False'; ExternalWritable := 'False'} : Bool;   // Activate standby "1"
         MovikitHandshakeIn { ExternalAccessible := 'False'; ExternalVisible := 'False'; ExternalWritable := 'False'} : Bool;   // If the MOVIKIT works the value will be copied into "MovikitHandshakeOut"
         EnableRapidStop { ExternalAccessible := 'False'; ExternalVisible := 'False'; ExternalWritable := 'False'} : Bool;   // Enable “1” / Rapid stop “0”
         EnableApplicationStop { ExternalAccessible := 'False'; ExternalVisible := 'False'; ExternalWritable := 'False'} : Bool;   // Enable “1” / Application stop “0”
         BIT_02_Reserved { ExternalAccessible := 'False'; ExternalVisible := 'False'; ExternalWritable := 'False'} : Bool;   // Reserved
         ReleaseBrake { ExternalAccessible := 'False'; ExternalVisible := 'False'; ExternalWritable := 'False'} : Bool;   // Release brake "1"
         JogPos { ExternalAccessible := 'False'; ExternalVisible := 'False'; ExternalWritable := 'False'} : Bool;   // Jog in positive direction "1"
         JogNeg { ExternalAccessible := 'False'; ExternalVisible := 'False'; ExternalWritable := 'False'} : Bool;   // Jog in negative direction "1"
         ApplyRelativePositioning { ExternalAccessible := 'False'; ExternalVisible := 'False'; ExternalWritable := 'False'} : Bool;   // Take the relative position from the FCB09 "1"
         StartStop { ExternalAccessible := 'False'; ExternalVisible := 'False'; ExternalWritable := 'False'} : Bool;   // Start "1" / Stop "0"
      END_STRUCT;
      SetpointSpeed : Int;   // Speed (Int) in rpm
      SetpointAcceleration : Int;   // Acceleration (Int) in rpm/s
      SetpointDeceleration : Int;   // Decceleration (Int) in rpm/s
   END_STRUCT;

END_TYPE

TYPE "UDT_VfdPositioningConfiguration"
TITLE = UDT_VfdPositioningConfiguration
VERSION : 0.1
//User defined stucture for configuring positioning device
   STRUCT
      TorqueMax : Real;   // VFD torque max - reference [Nm] as set up in SEW project
      SupplyFdbckOnDelayTime : UDInt;   // On delay time for supply feedback [ms]
      PositionWindow : DInt;   // Position window (tolerance) [mm]
      PositionMax : DInt;   // Maximum allowed position [mm]
      PositionMin : DInt;   // Minimum allowed position [mm]
      VFDSpeed : Int;   // Speed to run in automatic mode [mm/s]
      VFDAccDecel : Int;   // Acceleration and deceleration [mm/s2]
      VFDPNDeviceName : String;   // VFD's device name
      Position : Array[0..10] of DInt;   // Positions in mm to move to as requested
   END_STRUCT;

END_TYPE

TYPE "UDT_VfdSEWPositioningPI"
TITLE = UDT_VfdSEWPositioningPI
VERSION : 0.1
//User-defined structure of VFD SEW input telegram.
   STRUCT
      Status_Word_1 : Struct   // Status Word 1
         Error { ExternalAccessible := 'False'; ExternalVisible := 'False'; ExternalWritable := 'False'} : Bool;   // An error is active "1"
         Warning { ExternalAccessible := 'False'; ExternalVisible := 'False'; ExternalWritable := 'False'} : Bool;   // A warning is active "1"
         DriveTrain2Active { ExternalAccessible := 'False'; ExternalVisible := 'False'; ExternalWritable := 'False'} : Bool;   // Drive train 2 is active "1"
         VelocityTargetActualComparison { ExternalAccessible := 'False'; ExternalVisible := 'False'; ExternalWritable := 'False'} : Bool;   // The notification "Velocity target-actual-comparison" is on "1"
         SW_LimitSwitchInactive { ExternalAccessible := 'False'; ExternalVisible := 'False'; ExternalWritable := 'False'} : Bool;   // he software limit switch is inactive "1"
         BIT_13_Reserved { ExternalAccessible := 'False'; ExternalVisible := 'False'; ExternalWritable := 'False'} : Bool;   // Reserved
         StandbyActive { ExternalAccessible := 'False'; ExternalVisible := 'False'; ExternalWritable := 'False'} : Bool;   // Standby mode is active "1"
         MovikitHandshakeOut { ExternalAccessible := 'False'; ExternalVisible := 'False'; ExternalWritable := 'False'} : Bool;   // Copied value of "MovikitHandshakeIn"
         InverterReady { ExternalAccessible := 'False'; ExternalVisible := 'False'; ExternalWritable := 'False'} : Bool;   // There's no error and the inverter is ready "1"
         STO_Inactive { ExternalAccessible := 'False'; ExternalVisible := 'False'; ExternalWritable := 'False'} : Bool;   // STO is not active "1"
         OutputStageEnabled { ExternalAccessible := 'False'; ExternalVisible := 'False'; ExternalWritable := 'False'} : Bool;   // The output stage is released "1"
         BrakeReleased { ExternalAccessible := 'False'; ExternalVisible := 'False'; ExternalWritable := 'False'} : Bool;   // The brake is released "1"
         DriveActive { ExternalAccessible := 'False'; ExternalVisible := 'False'; ExternalWritable := 'False'} : Bool;   // The drive is active and the shaft turning "1"
         Referenced { ExternalAccessible := 'False'; ExternalVisible := 'False'; ExternalWritable := 'False'} : Bool;   // The drive is referenced "1"
         RelativePositionApplied { ExternalAccessible := 'False'; ExternalVisible := 'False'; ExternalWritable := 'False'} : Bool;   // The relative position is applied "1"
         InPosition { ExternalAccessible := 'False'; ExternalVisible := 'False'; ExternalWritable := 'False'} : Bool;   // The notification "in position" is on "1"
      END_STRUCT;
      ActualSpeed : Int;   // Actual drive speed (Int) [mm/s]
      StatusErrorNo : Word;   // Current status of the drive
      ActualTorque : Int;   // Actual torque in percent od the rated unit torque
      DigitalInput : Word;   // Digital inputs
      Mode : Int;   // Actual application mode (Int)
      ActualPosition_hW : Word;   // Actual position - High Word
      ActualPosition_lW : Word;   // Actual position - Low Word
   END_STRUCT;

END_TYPE

TYPE "UDT_ConveyorConfiguration"
TITLE = UDT_ConveyorConfiguration
VERSION : 0.1
//User-defined structure of conveyor parameters.
   STRUCT
      Common : "UDT_ConveyorCommonConfiguration";   // Common configuration
      Forward_Direction : Struct   // Forward Direction configuration
         EnergySaveLenght : DInt;   // Distance conveyor travelled before energy save activate [cm]
         GapHeadToHead : DInt;   // Gapping head to head value [cm]
         GapTailToHead : DInt;   // Gapping tail to head value [cm]
         GapCorrection : DInt;   // Gap offset to cover VFD's ramps [cm]
         PEC_EoSDistanceOffset : DInt;   // Distance offset between photo eye and the end of conveyor [mm]
         Mode : Int;   // Automatic operation; 1- Slave; 2- Queue;
         FirstConveyorToStart { ExternalAccessible := 'False'; ExternalVisible := 'False'; ExternalWritable := 'False'} : Bool;   // First conveyor to start cascade mode forward direction
      END_STRUCT;
      Reverse_Direction : Struct   // Reverse Direction configuration
         EnergySaveLenght : DInt;   // Distance conveyor travelled before energy save activate [cm]
         GapHeadToHead : DInt;   // Gapping head to head value [cm]
         GapTailToHead : DInt;   // Gapping tail to head value [cm]
         GapCorrection : DInt;   // Gap offset to cover VFD's ramps [cm]
         PEC_BoSDistanceOffset : DInt;   // Distance offset between photo eye and the end of conveyor [mm]
         Mode : Int;   // Automatic operation; 1- Slave; 2- Queue;
         FirstConveyorToStart { ExternalAccessible := 'False'; ExternalVisible := 'False'; ExternalWritable := 'False'} : Bool;   // First conveyor to start cascade mode reverse direction
      END_STRUCT;
      CascadeTimeOnDelay : UDInt;   // Cascade time on delay [ms]
      ExtraGapRecovery : DInt;   // Extra gap to recovery die back [cm]
      SpeedSetpointLow : Int;   // Low speed setpoint [mm/s]
      SpeedSetpointNominal : Int;   // Nominal speed setpoint [mm/s]
      Energy { ExternalAccessible := 'False'; ExternalVisible := 'False'; ExternalWritable := 'False'} : Bool;   // Energy save mode enable
      Bi_Directional_Enable { ExternalAccessible := 'False'; ExternalVisible := 'False'; ExternalWritable := 'False'} : Bool;   // The conveyor can run in both directions
   END_STRUCT;

END_TYPE

